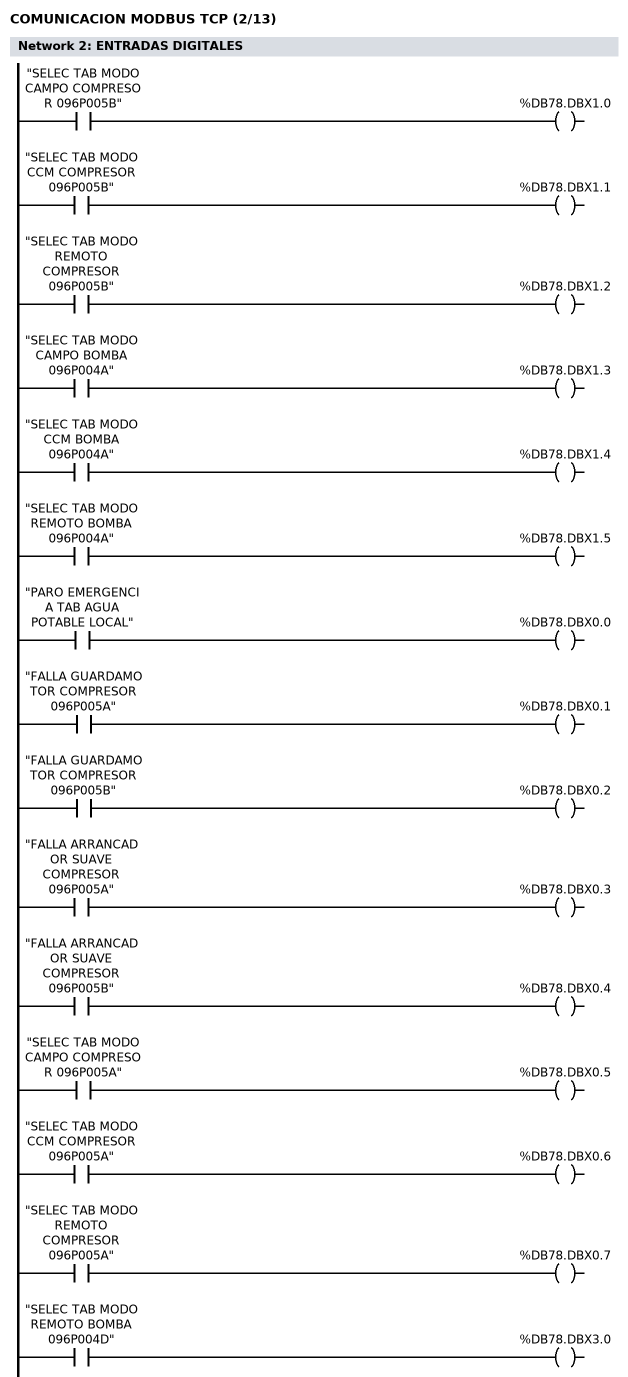
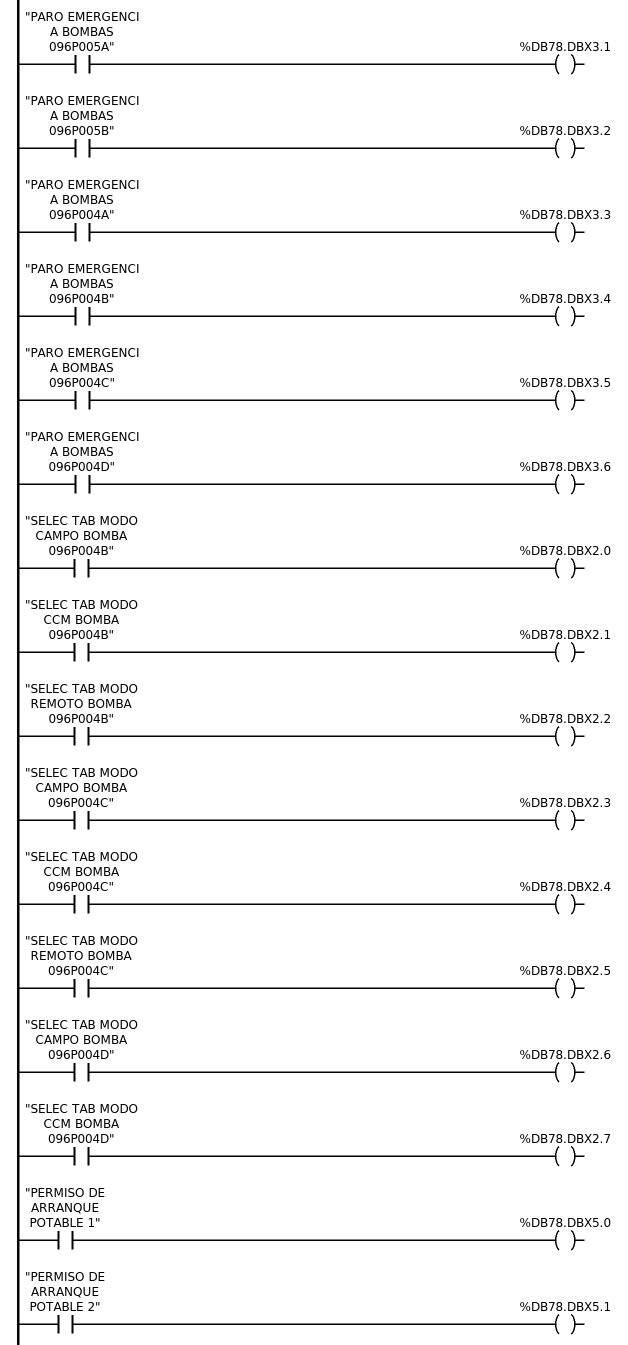
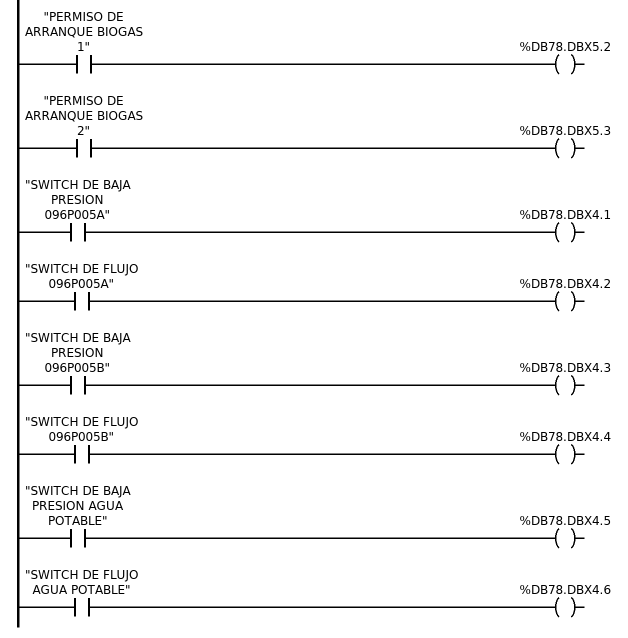
   RUNG wire#powerrail
      Contact( "SELEC TAB MODO CAMPO COMPRESOR 096P005B" )
      Coil( %DB78.DBX1.0 )
   END_RUNG
   RUNG wire#powerrail
      Contact( "SELEC TAB MODO CCM COMPRESOR 096P005B" )
      Coil( %DB78.DBX1.1 )
   END_RUNG
   RUNG wire#powerrail
      Contact( "SELEC TAB MODO REMOTO COMPRESOR 096P005B" )
      Coil( %DB78.DBX1.2 )
   END_RUNG
   RUNG wire#powerrail
      Contact( "SELEC TAB MODO CAMPO BOMBA 096P004A" )
      Coil( %DB78.DBX1.3 )
   END_RUNG
   RUNG wire#powerrail
      Contact( "SELEC TAB MODO CCM BOMBA 096P004A" )
      Coil( %DB78.DBX1.4 )
   END_RUNG
   RUNG wire#powerrail
      Contact( "SELEC TAB MODO REMOTO BOMBA 096P004A" )
      Coil( %DB78.DBX1.5 )
   END_RUNG
   RUNG wire#powerrail
      Contact( "PARO EMERGENCIA TAB AGUA POTABLE LOCAL" )
      Coil( %DB78.DBX0.0 )
   END_RUNG
   RUNG wire#powerrail
      Contact( "FALLA GUARDAMOTOR COMPRESOR 096P005A" )
      Coil( %DB78.DBX0.1 )
   END_RUNG
   RUNG wire#powerrail
      Contact( "FALLA GUARDAMOTOR COMPRESOR 096P005B" )
      Coil( %DB78.DBX0.2 )
   END_RUNG
   RUNG wire#powerrail
      Contact( "FALLA ARRANCADOR SUAVE COMPRESOR 096P005A" )
      Coil( %DB78.DBX0.3 )
   END_RUNG
   RUNG wire#powerrail
      Contact( "FALLA ARRANCADOR SUAVE COMPRESOR 096P005B" )
      Coil( %DB78.DBX0.4 )
   END_RUNG
   RUNG wire#powerrail
      Contact( "SELEC TAB MODO CAMPO COMPRESOR 096P005A" )
      Coil( %DB78.DBX0.5 )
   END_RUNG
   RUNG wire#powerrail
      Contact( "SELEC TAB MODO CCM COMPRESOR 096P005A" )
      Coil( %DB78.DBX0.6 )
   END_RUNG
   RUNG wire#powerrail
      Contact( "SELEC TAB MODO REMOTO COMPRESOR 096P005A" )
      Coil( %DB78.DBX0.7 )
   END_RUNG
   RUNG wire#powerrail
      Contact( "SELEC TAB MODO REMOTO BOMBA 096P004D" )
      Coil( %DB78.DBX3.0 )
   END_RUNG
   RUNG wire#powerrail
      Contact( "PARO EMERGENCIA BOMBAS 096P005A" )
      Coil( %DB78.DBX3.1 )
   END_RUNG
   RUNG wire#powerrail
      Contact( "PARO EMERGENCIA BOMBAS 096P005B" )
      Coil( %DB78.DBX3.2 )
   END_RUNG
   RUNG wire#powerrail
      Contact( "PARO EMERGENCIA BOMBAS 096P004A" )
      Coil( %DB78.DBX3.3 )
   END_RUNG
   RUNG wire#powerrail
      Contact( "PARO EMERGENCIA BOMBAS 096P004B" )
      Coil( %DB78.DBX3.4 )
   END_RUNG
   RUNG wire#powerrail
      Contact( "PARO EMERGENCIA BOMBAS 096P004C" )
      Coil( %DB78.DBX3.5 )
   END_RUNG
   RUNG wire#powerrail
      Contact( "PARO EMERGENCIA BOMBAS 096P004D" )
      Coil( %DB78.DBX3.6 )
   END_RUNG
   RUNG wire#powerrail
      Contact( "SELEC TAB MODO CAMPO BOMBA 096P004B" )
      Coil( %DB78.DBX2.0 )
   END_RUNG
   RUNG wire#powerrail
      Contact( "SELEC TAB MODO CCM BOMBA 096P004B" )
      Coil( %DB78.DBX2.1 )
   END_RUNG
   RUNG wire#powerrail
      Contact( "SELEC TAB MODO REMOTO BOMBA 096P004B" )
      Coil( %DB78.DBX2.2 )
   END_RUNG
   RUNG wire#powerrail
      Contact( "SELEC TAB MODO CAMPO BOMBA 096P004C" )
      Coil( %DB78.DBX2.3 )
   END_RUNG
   RUNG wire#powerrail
      Contact( "SELEC TAB MODO CCM BOMBA 096P004C" )
      Coil( %DB78.DBX2.4 )
   END_RUNG
   RUNG wire#powerrail
      Contact( "SELEC TAB MODO REMOTO BOMBA 096P004C" )
      Coil( %DB78.DBX2.5 )
   END_RUNG
   RUNG wire#powerrail
      Contact( "SELEC TAB MODO CAMPO BOMBA 096P004D" )
      Coil( %DB78.DBX2.6 )
   END_RUNG
   RUNG wire#powerrail
      Contact( "SELEC TAB MODO CCM BOMBA 096P004D" )
      Coil( %DB78.DBX2.7 )
   END_RUNG
   RUNG wire#powerrail
      Contact( "PERMISO DE ARRANQUE POTABLE 1" )
      Coil( %DB78.DBX5.0 )
   END_RUNG
   RUNG wire#powerrail
      Contact( "PERMISO DE ARRANQUE POTABLE 2" )
      Coil( %DB78.DBX5.1 )
   END_RUNG
   RUNG wire#powerrail
      Contact( "PERMISO DE ARRANQUE BIOGAS 1" )
      Coil( %DB78.DBX5.2 )
   END_RUNG
   RUNG wire#powerrail
      Contact( "PERMISO DE ARRANQUE BIOGAS 2" )
      Coil( %DB78.DBX5.3 )
   END_RUNG
   RUNG wire#powerrail
      Contact( "SWITCH DE BAJA PRESION 096P005A" )
      Coil( %DB78.DBX4.1 )
   END_RUNG
   RUNG wire#powerrail
      Contact( "SWITCH DE FLUJO 096P005A" )
      Coil( %DB78.DBX4.2 )
   END_RUNG
   RUNG wire#powerrail
      Contact( "SWITCH DE BAJA PRESION 096P005B" )
      Coil( %DB78.DBX4.3 )
   END_RUNG
   RUNG wire#powerrail
      Contact( "SWITCH DE FLUJO 096P005B" )
      Coil( %DB78.DBX4.4 )
   END_RUNG
   RUNG wire#powerrail
      Contact( "SWITCH DE BAJA PRESION AGUA POTABLE" )
      Coil( %DB78.DBX4.5 )
   END_RUNG
   RUNG wire#powerrail
      Contact( "SWITCH DE FLUJO AGUA POTABLE" )
      Coil( %DB78.DBX4.6 )
   END_RUNG
   // the same network as SCL:
   %DB78.DBX1.0 := "SELEC TAB MODO CAMPO COMPRESOR 096P005B";
   %DB78.DBX1.1 := "SELEC TAB MODO CCM COMPRESOR 096P005B";
   %DB78.DBX1.2 := "SELEC TAB MODO REMOTO COMPRESOR 096P005B";
   %DB78.DBX1.3 := "SELEC TAB MODO CAMPO BOMBA 096P004A";
   %DB78.DBX1.4 := "SELEC TAB MODO CCM BOMBA 096P004A";
   %DB78.DBX1.5 := "SELEC TAB MODO REMOTO BOMBA 096P004A";
   %DB78.DBX0.0 := "PARO EMERGENCIA TAB AGUA POTABLE LOCAL";
   %DB78.DBX0.1 := "FALLA GUARDAMOTOR COMPRESOR 096P005A";
   %DB78.DBX0.2 := "FALLA GUARDAMOTOR COMPRESOR 096P005B";
   %DB78.DBX0.3 := "FALLA ARRANCADOR SUAVE COMPRESOR 096P005A";
   %DB78.DBX0.4 := "FALLA ARRANCADOR SUAVE COMPRESOR 096P005B";
   %DB78.DBX0.5 := "SELEC TAB MODO CAMPO COMPRESOR 096P005A";
   %DB78.DBX0.6 := "SELEC TAB MODO CCM COMPRESOR 096P005A";
   %DB78.DBX0.7 := "SELEC TAB MODO REMOTO COMPRESOR 096P005A";
   %DB78.DBX3.0 := "SELEC TAB MODO REMOTO BOMBA 096P004D";
   %DB78.DBX3.1 := "PARO EMERGENCIA BOMBAS 096P005A";
   %DB78.DBX3.2 := "PARO EMERGENCIA BOMBAS 096P005B";
   %DB78.DBX3.3 := "PARO EMERGENCIA BOMBAS 096P004A";
   %DB78.DBX3.4 := "PARO EMERGENCIA BOMBAS 096P004B";
   %DB78.DBX3.5 := "PARO EMERGENCIA BOMBAS 096P004C";
   %DB78.DBX3.6 := "PARO EMERGENCIA BOMBAS 096P004D";
   %DB78.DBX2.0 := "SELEC TAB MODO CAMPO BOMBA 096P004B";
   %DB78.DBX2.1 := "SELEC TAB MODO CCM BOMBA 096P004B";
   %DB78.DBX2.2 := "SELEC TAB MODO REMOTO BOMBA 096P004B";
   %DB78.DBX2.3 := "SELEC TAB MODO CAMPO BOMBA 096P004C";
   %DB78.DBX2.4 := "SELEC TAB MODO CCM BOMBA 096P004C";
   %DB78.DBX2.5 := "SELEC TAB MODO REMOTO BOMBA 096P004C";
   %DB78.DBX2.6 := "SELEC TAB MODO CAMPO BOMBA 096P004D";
   %DB78.DBX2.7 := "SELEC TAB MODO CCM BOMBA 096P004D";
   %DB78.DBX5.0 := "PERMISO DE ARRANQUE POTABLE 1";
   %DB78.DBX5.1 := "PERMISO DE ARRANQUE POTABLE 2";
   %DB78.DBX5.2 := "PERMISO DE ARRANQUE BIOGAS 1";
   %DB78.DBX5.3 := "PERMISO DE ARRANQUE BIOGAS 2";
   %DB78.DBX4.1 := "SWITCH DE BAJA PRESION 096P005A";
   %DB78.DBX4.2 := "SWITCH DE FLUJO 096P005A";
   %DB78.DBX4.3 := "SWITCH DE BAJA PRESION 096P005B";
   %DB78.DBX4.4 := "SWITCH DE FLUJO 096P005B";
   %DB78.DBX4.5 := "SWITCH DE BAJA PRESION AGUA POTABLE";
   %DB78.DBX4.6 := "SWITCH DE FLUJO AGUA POTABLE";
END_REGION

REGION Network 3: SALIDAS DIGITALES
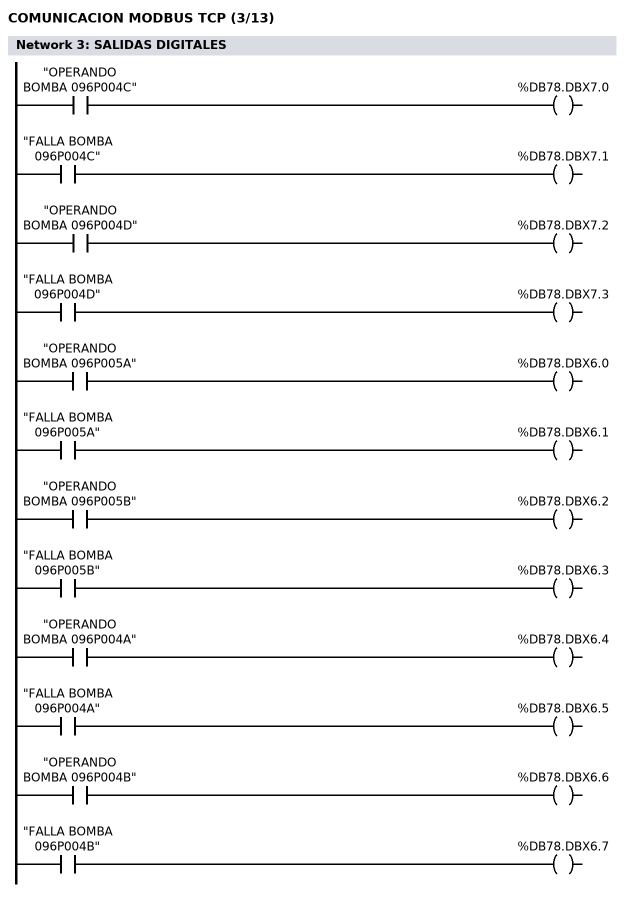
   RUNG wire#powerrail
      Contact( "OPERANDO BOMBA 096P004C" )
      Coil( %DB78.DBX7.0 )
   END_RUNG
   RUNG wire#powerrail
      Contact( "FALLA BOMBA 096P004C" )
      Coil( %DB78.DBX7.1 )
   END_RUNG
   RUNG wire#powerrail
      Contact( "OPERANDO BOMBA 096P004D" )
      Coil( %DB78.DBX7.2 )
   END_RUNG
   RUNG wire#powerrail
      Contact( "FALLA BOMBA 096P004D" )
      Coil( %DB78.DBX7.3 )
   END_RUNG
   RUNG wire#powerrail
      Contact( "OPERANDO BOMBA 096P005A" )
      Coil( %DB78.DBX6.0 )
   END_RUNG
   RUNG wire#powerrail
      Contact( "FALLA BOMBA 096P005A" )
      Coil( %DB78.DBX6.1 )
   END_RUNG
   RUNG wire#powerrail
      Contact( "OPERANDO BOMBA 096P005B" )
      Coil( %DB78.DBX6.2 )
   END_RUNG
   RUNG wire#powerrail
      Contact( "FALLA BOMBA 096P005B" )
      Coil( %DB78.DBX6.3 )
   END_RUNG
   RUNG wire#powerrail
      Contact( "OPERANDO BOMBA 096P004A" )
      Coil( %DB78.DBX6.4 )
   END_RUNG
   RUNG wire#powerrail
      Contact( "FALLA BOMBA 096P004A" )
      Coil( %DB78.DBX6.5 )
   END_RUNG
   RUNG wire#powerrail
      Contact( "OPERANDO BOMBA 096P004B" )
      Coil( %DB78.DBX6.6 )
   END_RUNG
   RUNG wire#powerrail
      Contact( "FALLA BOMBA 096P004B" )
      Coil( %DB78.DBX6.7 )
   END_RUNG
   // the same network as SCL:
   %DB78.DBX7.0 := "OPERANDO BOMBA 096P004C";
   %DB78.DBX7.1 := "FALLA BOMBA 096P004C";
   %DB78.DBX7.2 := "OPERANDO BOMBA 096P004D";
   %DB78.DBX7.3 := "FALLA BOMBA 096P004D";
   %DB78.DBX6.0 := "OPERANDO BOMBA 096P005A";
   %DB78.DBX6.1 := "FALLA BOMBA 096P005A";
   %DB78.DBX6.2 := "OPERANDO BOMBA 096P005B";
   %DB78.DBX6.3 := "FALLA BOMBA 096P005B";
   %DB78.DBX6.4 := "OPERANDO BOMBA 096P004A";
   %DB78.DBX6.5 := "FALLA BOMBA 096P004A";
   %DB78.DBX6.6 := "OPERANDO BOMBA 096P004B";
   %DB78.DBX6.7 := "FALLA BOMBA 096P004B";
END_REGION

REGION Network 4: SET POINT
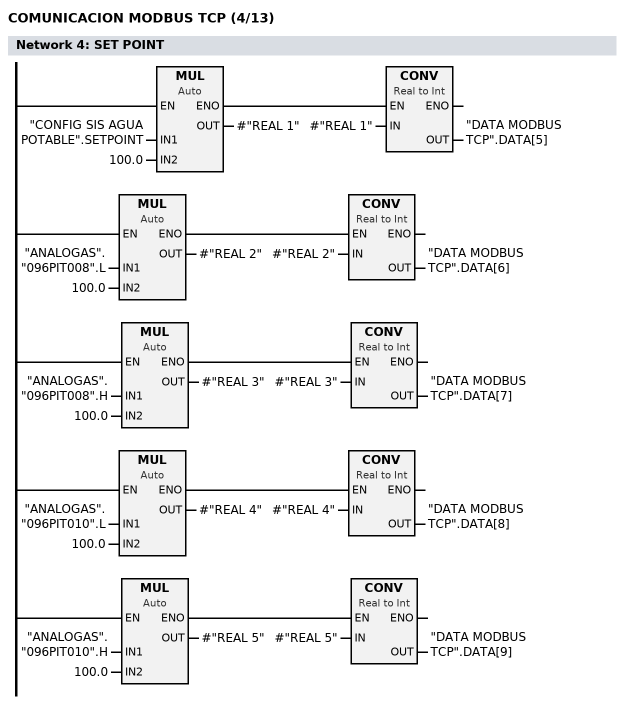
   RUNG wire#powerrail
      Mul(in1 := "CONFIG SIS AGUA POTABLE".SETPOINT, in2 := 100.0, out => #"REAL 1")
      { S7_Templates := "[SrcType := Real, DestType := Int]" } Convert(in := #"REAL 1", out => "DATA MODBUS TCP".DATA[5])
   END_RUNG
   RUNG wire#powerrail
      Mul(in1 := "ANALOGAS"."096PIT008".L, in2 := 100.0, out => #"REAL 2")
      { S7_Templates := "[SrcType := Real, DestType := Int]" } Convert(in := #"REAL 2", out => "DATA MODBUS TCP".DATA[6])
   END_RUNG
   RUNG wire#powerrail
      Mul(in1 := "ANALOGAS"."096PIT008".H, in2 := 100.0, out => #"REAL 3")
      { S7_Templates := "[SrcType := Real, DestType := Int]" } Convert(in := #"REAL 3", out => "DATA MODBUS TCP".DATA[7])
   END_RUNG
   RUNG wire#powerrail
      Mul(in1 := "ANALOGAS"."096PIT010".L, in2 := 100.0, out => #"REAL 4")
      { S7_Templates := "[SrcType := Real, DestType := Int]" } Convert(in := #"REAL 4", out => "DATA MODBUS TCP".DATA[8])
   END_RUNG
   RUNG wire#powerrail
      Mul(in1 := "ANALOGAS"."096PIT010".H, in2 := 100.0, out => #"REAL 5")
      { S7_Templates := "[SrcType := Real, DestType := Int]" } Convert(in := #"REAL 5", out => "DATA MODBUS TCP".DATA[9])
   END_RUNG
   // the same network as SCL:
   #"REAL 1" := "CONFIG SIS AGUA POTABLE".SETPOINT * 100.0;
   "DATA MODBUS TCP".DATA[5] := REAL_TO_INT(#"REAL 1");
   #"REAL 2" := "ANALOGAS"."096PIT008".L * 100.0;
   "DATA MODBUS TCP".DATA[6] := REAL_TO_INT(#"REAL 2");
   #"REAL 3" := "ANALOGAS"."096PIT008".H * 100.0;
   "DATA MODBUS TCP".DATA[7] := REAL_TO_INT(#"REAL 3");
   #"REAL 4" := "ANALOGAS"."096PIT010".L * 100.0;
   "DATA MODBUS TCP".DATA[8] := REAL_TO_INT(#"REAL 4");
   #"REAL 5" := "ANALOGAS"."096PIT010".H * 100.0;
   "DATA MODBUS TCP".DATA[9] := REAL_TO_INT(#"REAL 5");
END_REGION

REGION Network 5: ANALOGAS
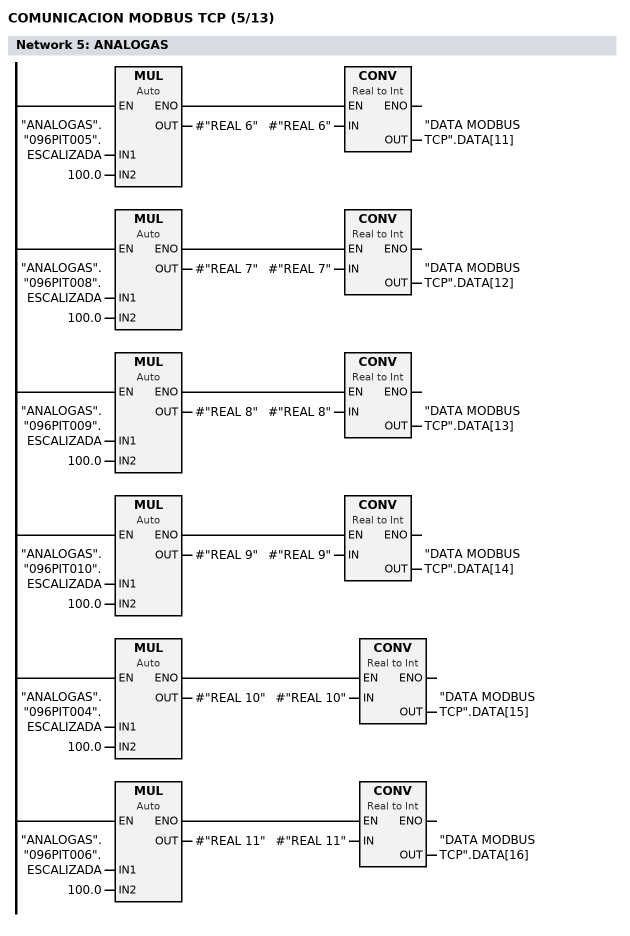
   RUNG wire#powerrail
      Mul(in1 := "ANALOGAS"."096PIT005".ESCALIZADA, in2 := 100.0, out => #"REAL 6")
      { S7_Templates := "[SrcType := Real, DestType := Int]" } Convert(in := #"REAL 6", out => "DATA MODBUS TCP".DATA[11])
   END_RUNG
   RUNG wire#powerrail
      Mul(in1 := "ANALOGAS"."096PIT008".ESCALIZADA, in2 := 100.0, out => #"REAL 7")
      { S7_Templates := "[SrcType := Real, DestType := Int]" } Convert(in := #"REAL 7", out => "DATA MODBUS TCP".DATA[12])
   END_RUNG
   RUNG wire#powerrail
      Mul(in1 := "ANALOGAS"."096PIT009".ESCALIZADA, in2 := 100.0, out => #"REAL 8")
      { S7_Templates := "[SrcType := Real, DestType := Int]" } Convert(in := #"REAL 8", out => "DATA MODBUS TCP".DATA[13])
   END_RUNG
   RUNG wire#powerrail
      Mul(in1 := "ANALOGAS"."096PIT010".ESCALIZADA, in2 := 100.0, out => #"REAL 9")
      { S7_Templates := "[SrcType := Real, DestType := Int]" } Convert(in := #"REAL 9", out => "DATA MODBUS TCP".DATA[14])
   END_RUNG
   RUNG wire#powerrail
      Mul(in1 := "ANALOGAS"."096PIT004".ESCALIZADA, in2 := 100.0, out => #"REAL 10")
      { S7_Templates := "[SrcType := Real, DestType := Int]" } Convert(in := #"REAL 10", out => "DATA MODBUS TCP".DATA[15])
   END_RUNG
   RUNG wire#powerrail
      Mul(in1 := "ANALOGAS"."096PIT006".ESCALIZADA, in2 := 100.0, out => #"REAL 11")
      { S7_Templates := "[SrcType := Real, DestType := Int]" } Convert(in := #"REAL 11", out => "DATA MODBUS TCP".DATA[16])
   END_RUNG
   // the same network as SCL:
   #"REAL 6" := "ANALOGAS"."096PIT005".ESCALIZADA * 100.0;
   "DATA MODBUS TCP".DATA[11] := REAL_TO_INT(#"REAL 6");
   #"REAL 7" := "ANALOGAS"."096PIT008".ESCALIZADA * 100.0;
   "DATA MODBUS TCP".DATA[12] := REAL_TO_INT(#"REAL 7");
   #"REAL 8" := "ANALOGAS"."096PIT009".ESCALIZADA * 100.0;
   "DATA MODBUS TCP".DATA[13] := REAL_TO_INT(#"REAL 8");
   #"REAL 9" := "ANALOGAS"."096PIT010".ESCALIZADA * 100.0;
   "DATA MODBUS TCP".DATA[14] := REAL_TO_INT(#"REAL 9");
   #"REAL 10" := "ANALOGAS"."096PIT004".ESCALIZADA * 100.0;
   "DATA MODBUS TCP".DATA[15] := REAL_TO_INT(#"REAL 10");
   #"REAL 11" := "ANALOGAS"."096PIT006".ESCALIZADA * 100.0;
   "DATA MODBUS TCP".DATA[16] := REAL_TO_INT(#"REAL 11");
END_REGION

REGION Network 6: ORDEN DE CAMBIO DE MODO BOMBA 5A
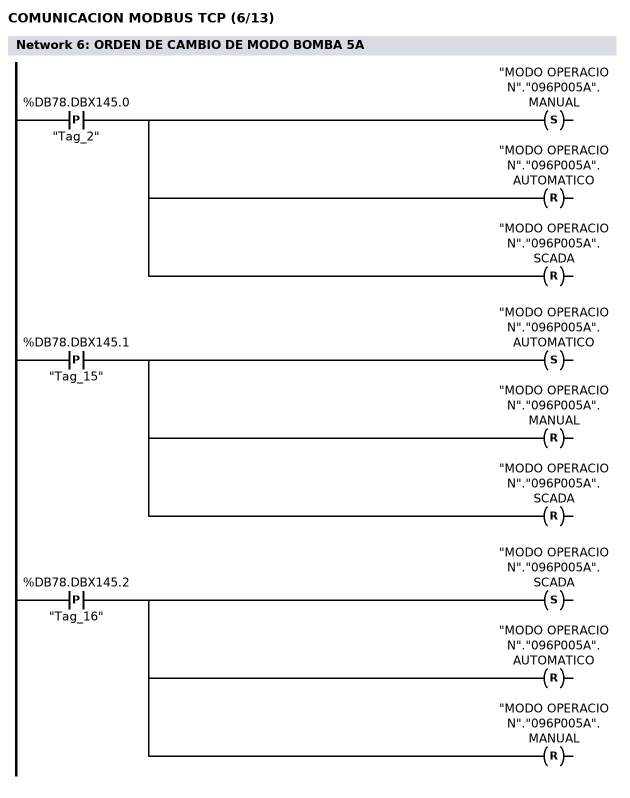
   RUNG wire#powerrail
      P_Contact(operand := %DB78.DBX145.0, bit := "Tag_2")
      wire#w1
      S_Coil( "MODO OPERACION"."096P005A".MANUAL )
   END_RUNG
   RUNG wire#w1
      R_Coil( "MODO OPERACION"."096P005A".AUTOMATICO )
   END_RUNG
   RUNG wire#w1
      R_Coil( "MODO OPERACION"."096P005A".SCADA )
   END_RUNG
   RUNG wire#powerrail
      P_Contact(operand := %DB78.DBX145.1, bit := "Tag_15")
      wire#w2
      S_Coil( "MODO OPERACION"."096P005A".AUTOMATICO )
   END_RUNG
   RUNG wire#w2
      R_Coil( "MODO OPERACION"."096P005A".MANUAL )
   END_RUNG
   RUNG wire#w2
      R_Coil( "MODO OPERACION"."096P005A".SCADA )
   END_RUNG
   RUNG wire#powerrail
      P_Contact(operand := %DB78.DBX145.2, bit := "Tag_16")
      wire#w3
      S_Coil( "MODO OPERACION"."096P005A".SCADA )
   END_RUNG
   RUNG wire#w3
      R_Coil( "MODO OPERACION"."096P005A".AUTOMATICO )
   END_RUNG
   RUNG wire#w3
      R_Coil( "MODO OPERACION"."096P005A".MANUAL )
   END_RUNG
   // the same network as SCL:
   #_w1 := %DB78.DBX145.0 AND NOT "Tag_2";   // rising edge of %DB78.DBX145.0
   "Tag_2" := %DB78.DBX145.0;
   IF #_w1 THEN
       "MODO OPERACION"."096P005A".MANUAL := TRUE;
       "MODO OPERACION"."096P005A".AUTOMATICO := FALSE;
       "MODO OPERACION"."096P005A".SCADA := FALSE;
   END_IF;
   #_w2 := %DB78.DBX145.1 AND NOT "Tag_15";   // rising edge of %DB78.DBX145.1
   "Tag_15" := %DB78.DBX145.1;
   IF #_w2 THEN
       "MODO OPERACION"."096P005A".AUTOMATICO := TRUE;
       "MODO OPERACION"."096P005A".MANUAL := FALSE;
       "MODO OPERACION"."096P005A".SCADA := FALSE;
   END_IF;
   #_w3 := %DB78.DBX145.2 AND NOT "Tag_16";   // rising edge of %DB78.DBX145.2
   "Tag_16" := %DB78.DBX145.2;
   IF #_w3 THEN
       "MODO OPERACION"."096P005A".SCADA := TRUE;
       "MODO OPERACION"."096P005A".AUTOMATICO := FALSE;
       "MODO OPERACION"."096P005A".MANUAL := FALSE;
   END_IF;
END_REGION

REGION Network 7: ORDEN DE CAMBIO DE MODO BOMBA 5B
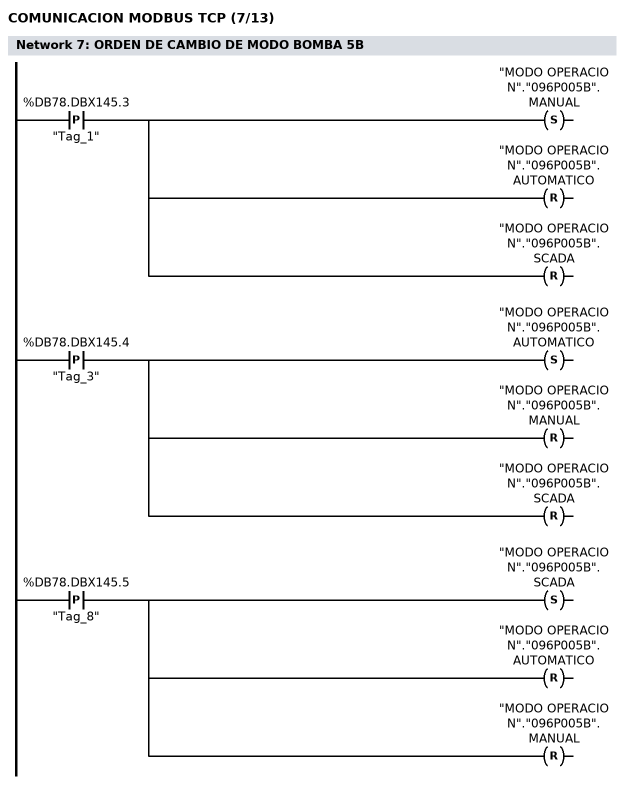
   RUNG wire#powerrail
      P_Contact(operand := %DB78.DBX145.3, bit := "Tag_1")
      wire#w1
      S_Coil( "MODO OPERACION"."096P005B".MANUAL )
   END_RUNG
   RUNG wire#w1
      R_Coil( "MODO OPERACION"."096P005B".AUTOMATICO )
   END_RUNG
   RUNG wire#w1
      R_Coil( "MODO OPERACION"."096P005B".SCADA )
   END_RUNG
   RUNG wire#powerrail
      P_Contact(operand := %DB78.DBX145.4, bit := "Tag_3")
      wire#w2
      S_Coil( "MODO OPERACION"."096P005B".AUTOMATICO )
   END_RUNG
   RUNG wire#w2
      R_Coil( "MODO OPERACION"."096P005B".MANUAL )
   END_RUNG
   RUNG wire#w2
      R_Coil( "MODO OPERACION"."096P005B".SCADA )
   END_RUNG
   RUNG wire#powerrail
      P_Contact(operand := %DB78.DBX145.5, bit := "Tag_8")
      wire#w3
      S_Coil( "MODO OPERACION"."096P005B".SCADA )
   END_RUNG
   RUNG wire#w3
      R_Coil( "MODO OPERACION"."096P005B".AUTOMATICO )
   END_RUNG
   RUNG wire#w3
      R_Coil( "MODO OPERACION"."096P005B".MANUAL )
   END_RUNG
   // the same network as SCL:
   #_w1 := %DB78.DBX145.3 AND NOT "Tag_1";   // rising edge of %DB78.DBX145.3
   "Tag_1" := %DB78.DBX145.3;
   IF #_w1 THEN
       "MODO OPERACION"."096P005B".MANUAL := TRUE;
       "MODO OPERACION"."096P005B".AUTOMATICO := FALSE;
       "MODO OPERACION"."096P005B".SCADA := FALSE;
   END_IF;
   #_w2 := %DB78.DBX145.4 AND NOT "Tag_3";   // rising edge of %DB78.DBX145.4
   "Tag_3" := %DB78.DBX145.4;
   IF #_w2 THEN
       "MODO OPERACION"."096P005B".AUTOMATICO := TRUE;
       "MODO OPERACION"."096P005B".MANUAL := FALSE;
       "MODO OPERACION"."096P005B".SCADA := FALSE;
   END_IF;
   #_w3 := %DB78.DBX145.5 AND NOT "Tag_8";   // rising edge of %DB78.DBX145.5
   "Tag_8" := %DB78.DBX145.5;
   IF #_w3 THEN
       "MODO OPERACION"."096P005B".SCADA := TRUE;
       "MODO OPERACION"."096P005B".AUTOMATICO := FALSE;
       "MODO OPERACION"."096P005B".MANUAL := FALSE;
   END_IF;
END_REGION

REGION Network 8: ORDEN DE CAMBIO DE MODO BOMBA 4A
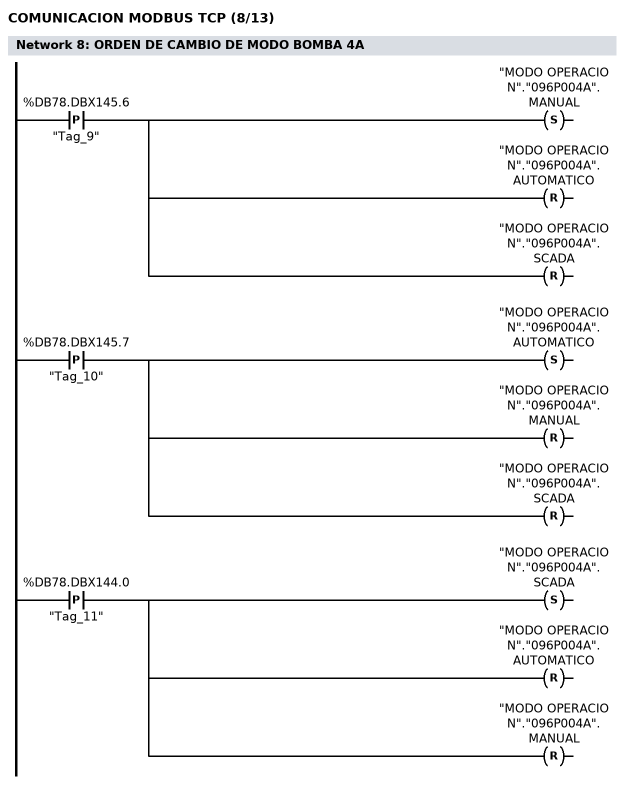
   RUNG wire#powerrail
      P_Contact(operand := %DB78.DBX145.6, bit := "Tag_9")
      wire#w1
      S_Coil( "MODO OPERACION"."096P004A".MANUAL )
   END_RUNG
   RUNG wire#w1
      R_Coil( "MODO OPERACION"."096P004A".AUTOMATICO )
   END_RUNG
   RUNG wire#w1
      R_Coil( "MODO OPERACION"."096P004A".SCADA )
   END_RUNG
   RUNG wire#powerrail
      P_Contact(operand := %DB78.DBX145.7, bit := "Tag_10")
      wire#w2
      S_Coil( "MODO OPERACION"."096P004A".AUTOMATICO )
   END_RUNG
   RUNG wire#w2
      R_Coil( "MODO OPERACION"."096P004A".MANUAL )
   END_RUNG
   RUNG wire#w2
      R_Coil( "MODO OPERACION"."096P004A".SCADA )
   END_RUNG
   RUNG wire#powerrail
      P_Contact(operand := %DB78.DBX144.0, bit := "Tag_11")
      wire#w3
      S_Coil( "MODO OPERACION"."096P004A".SCADA )
   END_RUNG
   RUNG wire#w3
      R_Coil( "MODO OPERACION"."096P004A".AUTOMATICO )
   END_RUNG
   RUNG wire#w3
      R_Coil( "MODO OPERACION"."096P004A".MANUAL )
   END_RUNG
   // the same network as SCL:
   #_w1 := %DB78.DBX145.6 AND NOT "Tag_9";   // rising edge of %DB78.DBX145.6
   "Tag_9" := %DB78.DBX145.6;
   IF #_w1 THEN
       "MODO OPERACION"."096P004A".MANUAL := TRUE;
       "MODO OPERACION"."096P004A".AUTOMATICO := FALSE;
       "MODO OPERACION"."096P004A".SCADA := FALSE;
   END_IF;
   #_w2 := %DB78.DBX145.7 AND NOT "Tag_10";   // rising edge of %DB78.DBX145.7
   "Tag_10" := %DB78.DBX145.7;
   IF #_w2 THEN
       "MODO OPERACION"."096P004A".AUTOMATICO := TRUE;
       "MODO OPERACION"."096P004A".MANUAL := FALSE;
       "MODO OPERACION"."096P004A".SCADA := FALSE;
   END_IF;
   #_w3 := %DB78.DBX144.0 AND NOT "Tag_11";   // rising edge of %DB78.DBX144.0
   "Tag_11" := %DB78.DBX144.0;
   IF #_w3 THEN
       "MODO OPERACION"."096P004A".SCADA := TRUE;
       "MODO OPERACION"."096P004A".AUTOMATICO := FALSE;
       "MODO OPERACION"."096P004A".MANUAL := FALSE;
   END_IF;
END_REGION

REGION Network 9: ORDEN DE CAMBIO DE MODO BOMBA 4B
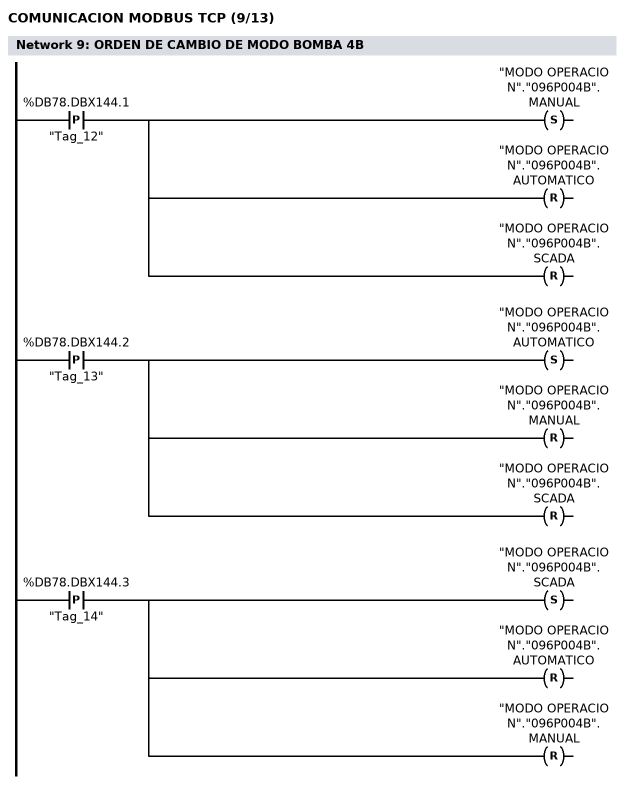
   RUNG wire#powerrail
      P_Contact(operand := %DB78.DBX144.1, bit := "Tag_12")
      wire#w1
      S_Coil( "MODO OPERACION"."096P004B".MANUAL )
   END_RUNG
   RUNG wire#w1
      R_Coil( "MODO OPERACION"."096P004B".AUTOMATICO )
   END_RUNG
   RUNG wire#w1
      R_Coil( "MODO OPERACION"."096P004B".SCADA )
   END_RUNG
   RUNG wire#powerrail
      P_Contact(operand := %DB78.DBX144.2, bit := "Tag_13")
      wire#w2
      S_Coil( "MODO OPERACION"."096P004B".AUTOMATICO )
   END_RUNG
   RUNG wire#w2
      R_Coil( "MODO OPERACION"."096P004B".MANUAL )
   END_RUNG
   RUNG wire#w2
      R_Coil( "MODO OPERACION"."096P004B".SCADA )
   END_RUNG
   RUNG wire#powerrail
      P_Contact(operand := %DB78.DBX144.3, bit := "Tag_14")
      wire#w3
      S_Coil( "MODO OPERACION"."096P004B".SCADA )
   END_RUNG
   RUNG wire#w3
      R_Coil( "MODO OPERACION"."096P004B".AUTOMATICO )
   END_RUNG
   RUNG wire#w3
      R_Coil( "MODO OPERACION"."096P004B".MANUAL )
   END_RUNG
   // the same network as SCL:
   #_w1 := %DB78.DBX144.1 AND NOT "Tag_12";   // rising edge of %DB78.DBX144.1
   "Tag_12" := %DB78.DBX144.1;
   IF #_w1 THEN
       "MODO OPERACION"."096P004B".MANUAL := TRUE;
       "MODO OPERACION"."096P004B".AUTOMATICO := FALSE;
       "MODO OPERACION"."096P004B".SCADA := FALSE;
   END_IF;
   #_w2 := %DB78.DBX144.2 AND NOT "Tag_13";   // rising edge of %DB78.DBX144.2
   "Tag_13" := %DB78.DBX144.2;
   IF #_w2 THEN
       "MODO OPERACION"."096P004B".AUTOMATICO := TRUE;
       "MODO OPERACION"."096P004B".MANUAL := FALSE;
       "MODO OPERACION"."096P004B".SCADA := FALSE;
   END_IF;
   #_w3 := %DB78.DBX144.3 AND NOT "Tag_14";   // rising edge of %DB78.DBX144.3
   "Tag_14" := %DB78.DBX144.3;
   IF #_w3 THEN
       "MODO OPERACION"."096P004B".SCADA := TRUE;
       "MODO OPERACION"."096P004B".AUTOMATICO := FALSE;
       "MODO OPERACION"."096P004B".MANUAL := FALSE;
   END_IF;
END_REGION

REGION Network 10: ORDEN DE CAMBIO DE MODO BOMBA 4C
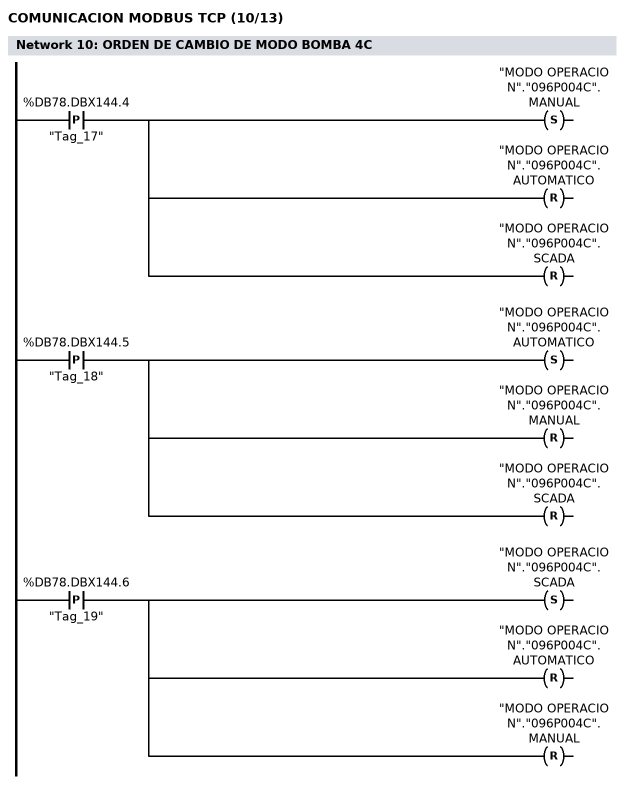
   RUNG wire#powerrail
      P_Contact(operand := %DB78.DBX144.4, bit := "Tag_17")
      wire#w1
      S_Coil( "MODO OPERACION"."096P004C".MANUAL )
   END_RUNG
   RUNG wire#w1
      R_Coil( "MODO OPERACION"."096P004C".AUTOMATICO )
   END_RUNG
   RUNG wire#w1
      R_Coil( "MODO OPERACION"."096P004C".SCADA )
   END_RUNG
   RUNG wire#powerrail
      P_Contact(operand := %DB78.DBX144.5, bit := "Tag_18")
      wire#w2
      S_Coil( "MODO OPERACION"."096P004C".AUTOMATICO )
   END_RUNG
   RUNG wire#w2
      R_Coil( "MODO OPERACION"."096P004C".MANUAL )
   END_RUNG
   RUNG wire#w2
      R_Coil( "MODO OPERACION"."096P004C".SCADA )
   END_RUNG
   RUNG wire#powerrail
      P_Contact(operand := %DB78.DBX144.6, bit := "Tag_19")
      wire#w3
      S_Coil( "MODO OPERACION"."096P004C".SCADA )
   END_RUNG
   RUNG wire#w3
      R_Coil( "MODO OPERACION"."096P004C".AUTOMATICO )
   END_RUNG
   RUNG wire#w3
      R_Coil( "MODO OPERACION"."096P004C".MANUAL )
   END_RUNG
   // the same network as SCL:
   #_w1 := %DB78.DBX144.4 AND NOT "Tag_17";   // rising edge of %DB78.DBX144.4
   "Tag_17" := %DB78.DBX144.4;
   IF #_w1 THEN
       "MODO OPERACION"."096P004C".MANUAL := TRUE;
       "MODO OPERACION"."096P004C".AUTOMATICO := FALSE;
       "MODO OPERACION"."096P004C".SCADA := FALSE;
   END_IF;
   #_w2 := %DB78.DBX144.5 AND NOT "Tag_18";   // rising edge of %DB78.DBX144.5
   "Tag_18" := %DB78.DBX144.5;
   IF #_w2 THEN
       "MODO OPERACION"."096P004C".AUTOMATICO := TRUE;
       "MODO OPERACION"."096P004C".MANUAL := FALSE;
       "MODO OPERACION"."096P004C".SCADA := FALSE;
   END_IF;
   #_w3 := %DB78.DBX144.6 AND NOT "Tag_19";   // rising edge of %DB78.DBX144.6
   "Tag_19" := %DB78.DBX144.6;
   IF #_w3 THEN
       "MODO OPERACION"."096P004C".SCADA := TRUE;
       "MODO OPERACION"."096P004C".AUTOMATICO := FALSE;
       "MODO OPERACION"."096P004C".MANUAL := FALSE;
   END_IF;
END_REGION

REGION Network 11: ORDEN DE CAMBIO DE MODO BOMBA 4D
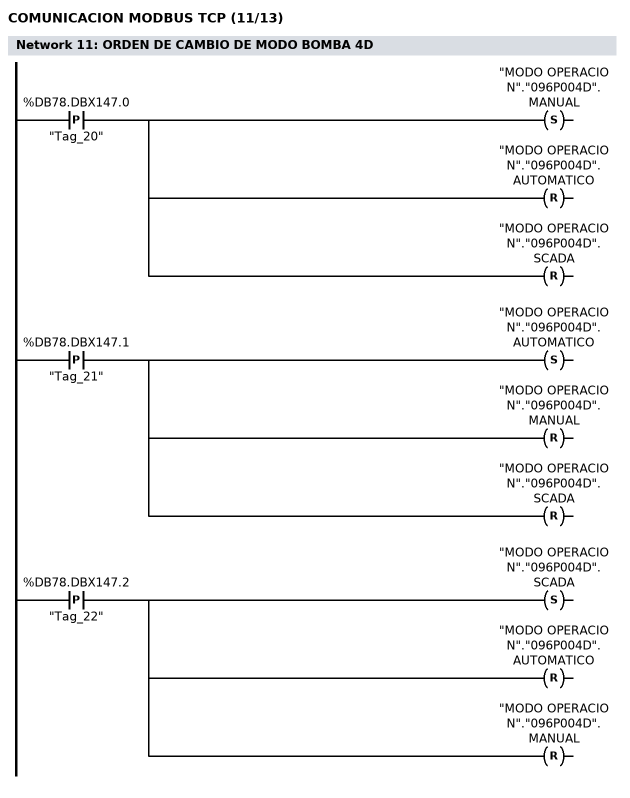
   RUNG wire#powerrail
      P_Contact(operand := %DB78.DBX147.0, bit := "Tag_20")
      wire#w1
      S_Coil( "MODO OPERACION"."096P004D".MANUAL )
   END_RUNG
   RUNG wire#w1
      R_Coil( "MODO OPERACION"."096P004D".AUTOMATICO )
   END_RUNG
   RUNG wire#w1
      R_Coil( "MODO OPERACION"."096P004D".SCADA )
   END_RUNG
   RUNG wire#powerrail
      P_Contact(operand := %DB78.DBX147.1, bit := "Tag_21")
      wire#w2
      S_Coil( "MODO OPERACION"."096P004D".AUTOMATICO )
   END_RUNG
   RUNG wire#w2
      R_Coil( "MODO OPERACION"."096P004D".MANUAL )
   END_RUNG
   RUNG wire#w2
      R_Coil( "MODO OPERACION"."096P004D".SCADA )
   END_RUNG
   RUNG wire#powerrail
      P_Contact(operand := %DB78.DBX147.2, bit := "Tag_22")
      wire#w3
      S_Coil( "MODO OPERACION"."096P004D".SCADA )
   END_RUNG
   RUNG wire#w3
      R_Coil( "MODO OPERACION"."096P004D".AUTOMATICO )
   END_RUNG
   RUNG wire#w3
      R_Coil( "MODO OPERACION"."096P004D".MANUAL )
   END_RUNG
   // the same network as SCL:
   #_w1 := %DB78.DBX147.0 AND NOT "Tag_20";   // rising edge of %DB78.DBX147.0
   "Tag_20" := %DB78.DBX147.0;
   IF #_w1 THEN
       "MODO OPERACION"."096P004D".MANUAL := TRUE;
       "MODO OPERACION"."096P004D".AUTOMATICO := FALSE;
       "MODO OPERACION"."096P004D".SCADA := FALSE;
   END_IF;
   #_w2 := %DB78.DBX147.1 AND NOT "Tag_21";   // rising edge of %DB78.DBX147.1
   "Tag_21" := %DB78.DBX147.1;
   IF #_w2 THEN
       "MODO OPERACION"."096P004D".AUTOMATICO := TRUE;
       "MODO OPERACION"."096P004D".MANUAL := FALSE;
       "MODO OPERACION"."096P004D".SCADA := FALSE;
   END_IF;
   #_w3 := %DB78.DBX147.2 AND NOT "Tag_22";   // rising edge of %DB78.DBX147.2
   "Tag_22" := %DB78.DBX147.2;
   IF #_w3 THEN
       "MODO OPERACION"."096P004D".SCADA := TRUE;
       "MODO OPERACION"."096P004D".AUTOMATICO := FALSE;
       "MODO OPERACION"."096P004D".MANUAL := FALSE;
   END_IF;
END_REGION

REGION Network 12: estados modos de operacion
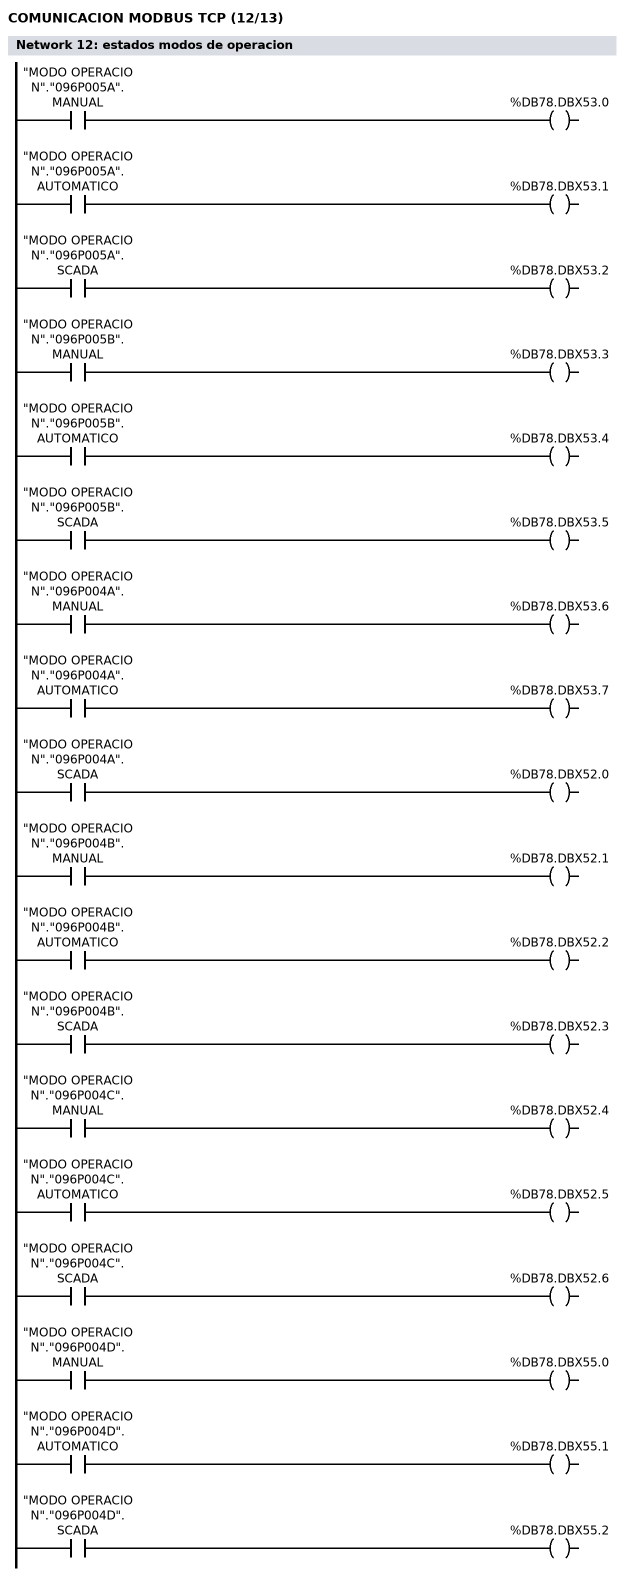
   RUNG wire#powerrail
      Contact( "MODO OPERACION"."096P005A".MANUAL )
      Coil( %DB78.DBX53.0 )
   END_RUNG
   RUNG wire#powerrail
      Contact( "MODO OPERACION"."096P005A".AUTOMATICO )
      Coil( %DB78.DBX53.1 )
   END_RUNG
   RUNG wire#powerrail
      Contact( "MODO OPERACION"."096P005A".SCADA )
      Coil( %DB78.DBX53.2 )
   END_RUNG
   RUNG wire#powerrail
      Contact( "MODO OPERACION"."096P005B".MANUAL )
      Coil( %DB78.DBX53.3 )
   END_RUNG
   RUNG wire#powerrail
      Contact( "MODO OPERACION"."096P005B".AUTOMATICO )
      Coil( %DB78.DBX53.4 )
   END_RUNG
   RUNG wire#powerrail
      Contact( "MODO OPERACION"."096P005B".SCADA )
      Coil( %DB78.DBX53.5 )
   END_RUNG
   RUNG wire#powerrail
      Contact( "MODO OPERACION"."096P004A".MANUAL )
      Coil( %DB78.DBX53.6 )
   END_RUNG
   RUNG wire#powerrail
      Contact( "MODO OPERACION"."096P004A".AUTOMATICO )
      Coil( %DB78.DBX53.7 )
   END_RUNG
   RUNG wire#powerrail
      Contact( "MODO OPERACION"."096P004A".SCADA )
      Coil( %DB78.DBX52.0 )
   END_RUNG
   RUNG wire#powerrail
      Contact( "MODO OPERACION"."096P004B".MANUAL )
      Coil( %DB78.DBX52.1 )
   END_RUNG
   RUNG wire#powerrail
      Contact( "MODO OPERACION"."096P004B".AUTOMATICO )
      Coil( %DB78.DBX52.2 )
   END_RUNG
   RUNG wire#powerrail
      Contact( "MODO OPERACION"."096P004B".SCADA )
      Coil( %DB78.DBX52.3 )
   END_RUNG
   RUNG wire#powerrail
      Contact( "MODO OPERACION"."096P004C".MANUAL )
      Coil( %DB78.DBX52.4 )
   END_RUNG
   RUNG wire#powerrail
      Contact( "MODO OPERACION"."096P004C".AUTOMATICO )
      Coil( %DB78.DBX52.5 )
   END_RUNG
   RUNG wire#powerrail
      Contact( "MODO OPERACION"."096P004C".SCADA )
      Coil( %DB78.DBX52.6 )
   END_RUNG
   RUNG wire#powerrail
      Contact( "MODO OPERACION"."096P004D".MANUAL )
      Coil( %DB78.DBX55.0 )
   END_RUNG
   RUNG wire#powerrail
      Contact( "MODO OPERACION"."096P004D".AUTOMATICO )
      Coil( %DB78.DBX55.1 )
   END_RUNG
   RUNG wire#powerrail
      Contact( "MODO OPERACION"."096P004D".SCADA )
      Coil( %DB78.DBX55.2 )
   END_RUNG
   // the same network as SCL:
   %DB78.DBX53.0 := "MODO OPERACION"."096P005A".MANUAL;
   %DB78.DBX53.1 := "MODO OPERACION"."096P005A".AUTOMATICO;
   %DB78.DBX53.2 := "MODO OPERACION"."096P005A".SCADA;
   %DB78.DBX53.3 := "MODO OPERACION"."096P005B".MANUAL;
   %DB78.DBX53.4 := "MODO OPERACION"."096P005B".AUTOMATICO;
   %DB78.DBX53.5 := "MODO OPERACION"."096P005B".SCADA;
   %DB78.DBX53.6 := "MODO OPERACION"."096P004A".MANUAL;
   %DB78.DBX53.7 := "MODO OPERACION"."096P004A".AUTOMATICO;
   %DB78.DBX52.0 := "MODO OPERACION"."096P004A".SCADA;
   %DB78.DBX52.1 := "MODO OPERACION"."096P004B".MANUAL;
   %DB78.DBX52.2 := "MODO OPERACION"."096P004B".AUTOMATICO;
   %DB78.DBX52.3 := "MODO OPERACION"."096P004B".SCADA;
   %DB78.DBX52.4 := "MODO OPERACION"."096P004C".MANUAL;
   %DB78.DBX52.5 := "MODO OPERACION"."096P004C".AUTOMATICO;
   %DB78.DBX52.6 := "MODO OPERACION"."096P004C".SCADA;
   %DB78.DBX55.0 := "MODO OPERACION"."096P004D".MANUAL;
   %DB78.DBX55.1 := "MODO OPERACION"."096P004D".AUTOMATICO;
   %DB78.DBX55.2 := "MODO OPERACION"."096P004D".SCADA;
END_REGION

REGION Network 13: ESTADO VFDS
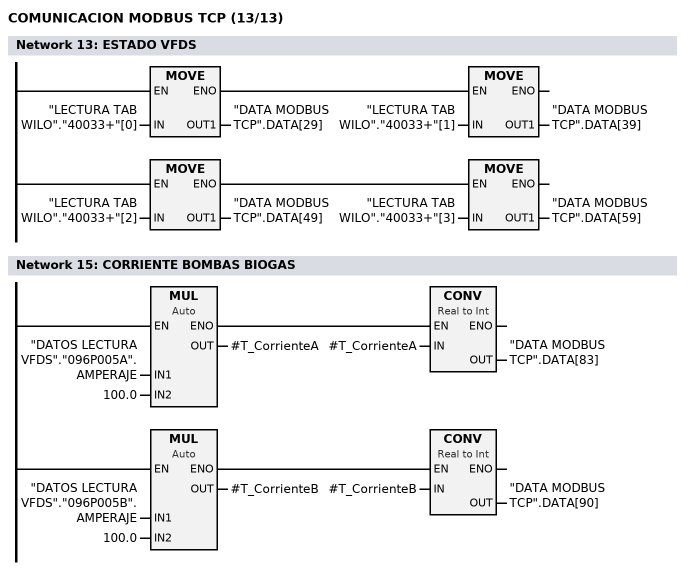
   RUNG wire#powerrail
      Move(in := "LECTURA TAB WILO"."40033+"[0], out1 => "DATA MODBUS TCP".DATA[29])
      Move(in := "LECTURA TAB WILO"."40033+"[1], out1 => "DATA MODBUS TCP".DATA[39])
   END_RUNG
   RUNG wire#powerrail
      Move(in := "LECTURA TAB WILO"."40033+"[2], out1 => "DATA MODBUS TCP".DATA[49])
      Move(in := "LECTURA TAB WILO"."40033+"[3], out1 => "DATA MODBUS TCP".DATA[59])
   END_RUNG
   // the same network as SCL:
   "DATA MODBUS TCP".DATA[29] := "LECTURA TAB WILO"."40033+"[0];
   "DATA MODBUS TCP".DATA[39] := "LECTURA TAB WILO"."40033+"[1];
   "DATA MODBUS TCP".DATA[49] := "LECTURA TAB WILO"."40033+"[2];
   "DATA MODBUS TCP".DATA[59] := "LECTURA TAB WILO"."40033+"[3];
END_REGION

REGION Network 15: CORRIENTE BOMBAS BIOGAS
   RUNG wire#powerrail
      Mul(in1 := "DATOS LECTURA VFDS"."096P005A".AMPERAJE, in2 := 100.0, out => #T_CorrienteA)
      { S7_Templates := "[SrcType := Real, DestType := Int]" } Convert(in := #T_CorrienteA, out => "DATA MODBUS TCP".DATA[83])
   END_RUNG
   RUNG wire#powerrail
      Mul(in1 := "DATOS LECTURA VFDS"."096P005B".AMPERAJE, in2 := 100.0, out => #T_CorrienteB)
      { S7_Templates := "[SrcType := Real, DestType := Int]" } Convert(in := #T_CorrienteB, out => "DATA MODBUS TCP".DATA[90])
   END_RUNG
   // the same network as SCL:
   #T_CorrienteA := "DATOS LECTURA VFDS"."096P005A".AMPERAJE * 100.0;
   "DATA MODBUS TCP".DATA[83] := REAL_TO_INT(#T_CorrienteA);
   #T_CorrienteB := "DATOS LECTURA VFDS"."096P005B".AMPERAJE * 100.0;
   "DATA MODBUS TCP".DATA[90] := REAL_TO_INT(#T_CorrienteB);
END_REGION
END_FUNCTION

FUNCTION "Comunicacion RTU" : Void   // FC8, LAD
{ S7_Optimized_Access := 'TRUE' }
VERSION : 0.1
   VAR_TEMP
      "RESET TEMP" : Bool;
      TEST1 : Bool;
   END_VAR
BEGIN

REGION Network 1: CONTEO COMUNICACION
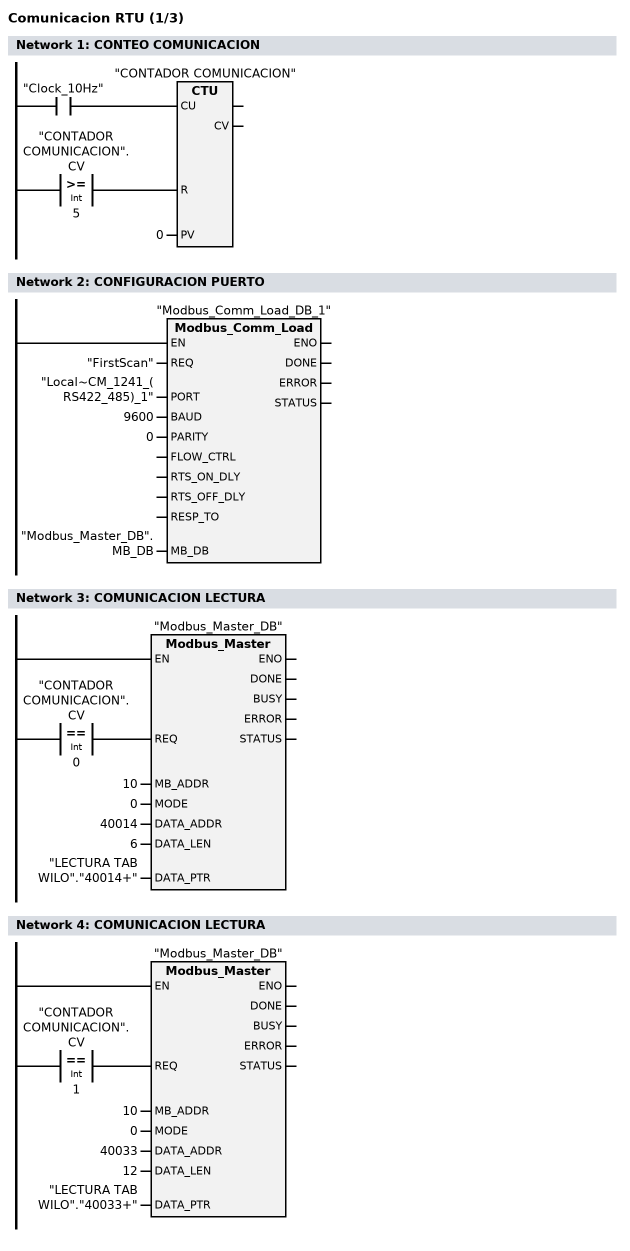
   "CONTADOR COMUNICACION".CTU(CU := "Clock_10Hz", R := "CONTADOR COMUNICACION".CV >= 5, PV := 0);
END_REGION

REGION Network 2: CONFIGURACION PUERTO
   "Modbus_Comm_Load_DB_1"(REQ := "FirstScan",   // Modbus_Comm_Load
                           PORT := "Local~CM_1241_(RS422_485)_1",
                           BAUD := 9600,
                           PARITY := 0,
                           MB_DB := "Modbus_Master_DB".MB_DB);
END_REGION

REGION Network 3: COMUNICACION LECTURA
   "Modbus_Master_DB"(REQ := "CONTADOR COMUNICACION".CV = 0,   // Modbus_Master
                      MB_ADDR := 10,
                      MODE := 0,
                      DATA_ADDR := 40014,
                      DATA_LEN := 6,
                      DATA_PTR := "LECTURA TAB WILO"."40014+");
END_REGION

REGION Network 4: COMUNICACION LECTURA
   "Modbus_Master_DB"(REQ := "CONTADOR COMUNICACION".CV = 1,   // Modbus_Master
                      MB_ADDR := 10,
                      MODE := 0,
                      DATA_ADDR := 40033,
                      DATA_LEN := 12,
                      DATA_PTR := "LECTURA TAB WILO"."40033+");
END_REGION

REGION Network 5: COMUNICACION LECTURA
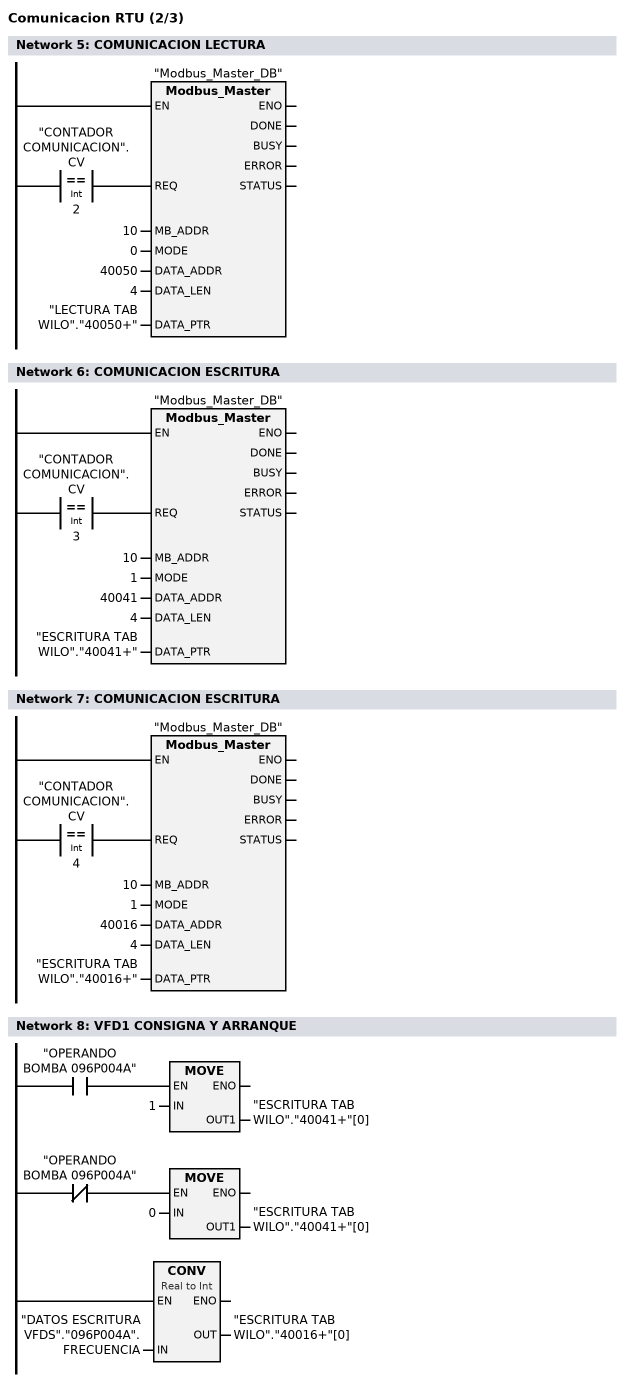
   "Modbus_Master_DB"(REQ := "CONTADOR COMUNICACION".CV = 2,   // Modbus_Master
                      MB_ADDR := 10,
                      MODE := 0,
                      DATA_ADDR := 40050,
                      DATA_LEN := 4,
                      DATA_PTR := "LECTURA TAB WILO"."40050+");
END_REGION

REGION Network 6: COMUNICACION ESCRITURA
   "Modbus_Master_DB"(REQ := "CONTADOR COMUNICACION".CV = 3,   // Modbus_Master
                      MB_ADDR := 10,
                      MODE := 1,
                      DATA_ADDR := 40041,
                      DATA_LEN := 4,
                      DATA_PTR := "ESCRITURA TAB WILO"."40041+");
END_REGION

REGION Network 7: COMUNICACION ESCRITURA
   "Modbus_Master_DB"(REQ := "CONTADOR COMUNICACION".CV = 4,   // Modbus_Master
                      MB_ADDR := 10,
                      MODE := 1,
                      DATA_ADDR := 40016,
                      DATA_LEN := 4,
                      DATA_PTR := "ESCRITURA TAB WILO"."40016+");
END_REGION

REGION Network 8: VFD1 CONSIGNA Y ARRANQUE
   RUNG wire#powerrail
      Contact( "OPERANDO BOMBA 096P004A" )
      Move(in := 1, out1 => "ESCRITURA TAB WILO"."40041+"[0])
   END_RUNG
   RUNG wire#powerrail
      I_Contact( "OPERANDO BOMBA 096P004A" )
      Move(in := 0, out1 => "ESCRITURA TAB WILO"."40041+"[0])
   END_RUNG
   RUNG wire#powerrail
      { S7_Templates := "[SrcType := Real, DestType := Int]" } Convert(in := "DATOS ESCRITURA VFDS"."096P004A".FRECUENCIA, out => "ESCRITURA TAB WILO"."40016+"[0])
   END_RUNG
   // the same network as SCL:
   IF "OPERANDO BOMBA 096P004A" THEN "ESCRITURA TAB WILO"."40041+"[0] := 1; END_IF;
   IF NOT "OPERANDO BOMBA 096P004A" THEN "ESCRITURA TAB WILO"."40041+"[0] := 0; END_IF;
   "ESCRITURA TAB WILO"."40016+"[0] := REAL_TO_INT("DATOS ESCRITURA VFDS"."096P004A".FRECUENCIA);
END_REGION

REGION Network 9: VFD2 CONSIGNA Y ARRANQUE
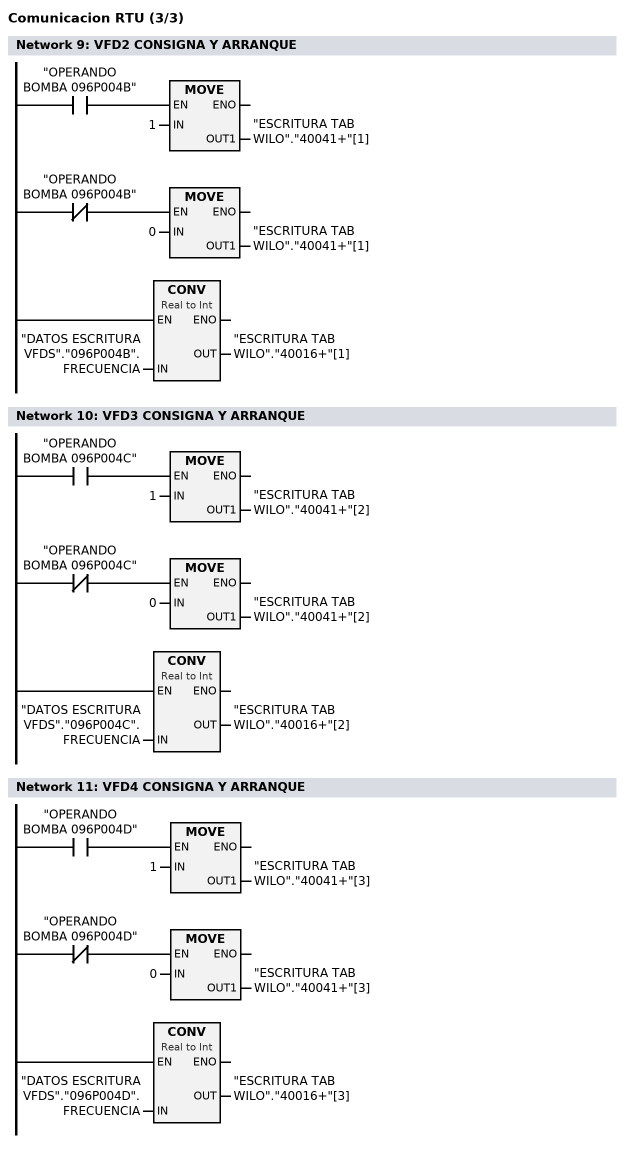
   RUNG wire#powerrail
      Contact( "OPERANDO BOMBA 096P004B" )
      Move(in := 1, out1 => "ESCRITURA TAB WILO"."40041+"[1])
   END_RUNG
   RUNG wire#powerrail
      I_Contact( "OPERANDO BOMBA 096P004B" )
      Move(in := 0, out1 => "ESCRITURA TAB WILO"."40041+"[1])
   END_RUNG
   RUNG wire#powerrail
      { S7_Templates := "[SrcType := Real, DestType := Int]" } Convert(in := "DATOS ESCRITURA VFDS"."096P004B".FRECUENCIA, out => "ESCRITURA TAB WILO"."40016+"[1])
   END_RUNG
   // the same network as SCL:
   IF "OPERANDO BOMBA 096P004B" THEN "ESCRITURA TAB WILO"."40041+"[1] := 1; END_IF;
   IF NOT "OPERANDO BOMBA 096P004B" THEN "ESCRITURA TAB WILO"."40041+"[1] := 0; END_IF;
   "ESCRITURA TAB WILO"."40016+"[1] := REAL_TO_INT("DATOS ESCRITURA VFDS"."096P004B".FRECUENCIA);
END_REGION

REGION Network 10: VFD3 CONSIGNA Y ARRANQUE
   RUNG wire#powerrail
      Contact( "OPERANDO BOMBA 096P004C" )
      Move(in := 1, out1 => "ESCRITURA TAB WILO"."40041+"[2])
   END_RUNG
   RUNG wire#powerrail
      I_Contact( "OPERANDO BOMBA 096P004C" )
      Move(in := 0, out1 => "ESCRITURA TAB WILO"."40041+"[2])
   END_RUNG
   RUNG wire#powerrail
      { S7_Templates := "[SrcType := Real, DestType := Int]" } Convert(in := "DATOS ESCRITURA VFDS"."096P004C".FRECUENCIA, out => "ESCRITURA TAB WILO"."40016+"[2])
   END_RUNG
   // the same network as SCL:
   IF "OPERANDO BOMBA 096P004C" THEN "ESCRITURA TAB WILO"."40041+"[2] := 1; END_IF;
   IF NOT "OPERANDO BOMBA 096P004C" THEN "ESCRITURA TAB WILO"."40041+"[2] := 0; END_IF;
   "ESCRITURA TAB WILO"."40016+"[2] := REAL_TO_INT("DATOS ESCRITURA VFDS"."096P004C".FRECUENCIA);
END_REGION

REGION Network 11: VFD4 CONSIGNA Y ARRANQUE
   RUNG wire#powerrail
      Contact( "OPERANDO BOMBA 096P004D" )
      Move(in := 1, out1 => "ESCRITURA TAB WILO"."40041+"[3])
   END_RUNG
   RUNG wire#powerrail
      I_Contact( "OPERANDO BOMBA 096P004D" )
      Move(in := 0, out1 => "ESCRITURA TAB WILO"."40041+"[3])
   END_RUNG
   RUNG wire#powerrail
      { S7_Templates := "[SrcType := Real, DestType := Int]" } Convert(in := "DATOS ESCRITURA VFDS"."096P004D".FRECUENCIA, out => "ESCRITURA TAB WILO"."40016+"[3])
   END_RUNG
   // the same network as SCL:
   IF "OPERANDO BOMBA 096P004D" THEN "ESCRITURA TAB WILO"."40041+"[3] := 1; END_IF;
   IF NOT "OPERANDO BOMBA 096P004D" THEN "ESCRITURA TAB WILO"."40041+"[3] := 0; END_IF;
   "ESCRITURA TAB WILO"."40016+"[3] := REAL_TO_INT("DATOS ESCRITURA VFDS"."096P004D".FRECUENCIA);
END_REGION
END_FUNCTION

FUNCTION "DATOS HMI" : Void   // FC9, LAD
{ S7_Optimized_Access := 'TRUE' }
VERSION : 0.1
   VAR_TEMP
      "FRECUENCIA 1" : Real;
      "FRECUENCIA 2" : Real;
      "FRECUENCIA 3" : Real;
      "FRECUENCIA 4" : Real;
   END_VAR
BEGIN

REGION Network 1: VFD1
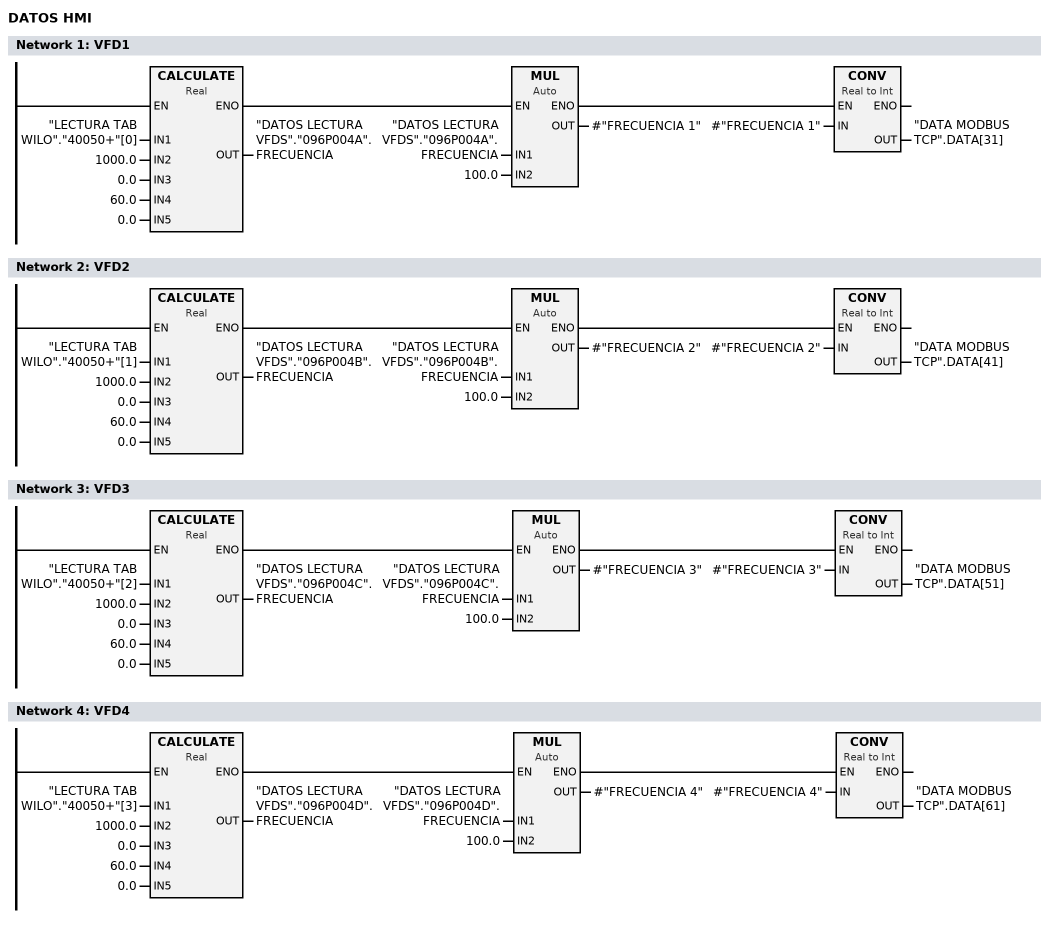
   RUNG wire#powerrail
      { S7_Templates := "SrcType := Real"; S7_Expression := "(((IN4-IN5)/(IN2-IN3))*IN1)+(IN5-(((IN4-IN5)/(IN2-IN3))*IN3))" } Calculate(in1 := "LECTURA TAB WILO"."40050+"[0], in2 := 1000.0, in3 := 0.0, in4 := 60.0, in5 := 0.0, out => "DATOS LECTURA VFDS"."096P004A".FRECUENCIA)
      Mul(in1 := "DATOS LECTURA VFDS"."096P004A".FRECUENCIA, in2 := 100.0, out => #"FRECUENCIA 1")
      { S7_Templates := "[SrcType := Real, DestType := Int]" } Convert(in := #"FRECUENCIA 1", out => "DATA MODBUS TCP".DATA[31])
   END_RUNG
   // the same network as SCL:
   "DATOS LECTURA VFDS"."096P004A".FRECUENCIA := (((60.0-0.0)/(1000.0-0.0))*"LECTURA TAB WILO"."40050+"[0])+(0.0-(((60.0-0.0)/(1000.0-0.0))*0.0));
   #"FRECUENCIA 1" := "DATOS LECTURA VFDS"."096P004A".FRECUENCIA * 100.0;
   "DATA MODBUS TCP".DATA[31] := REAL_TO_INT(#"FRECUENCIA 1");
END_REGION

REGION Network 2: VFD2
   RUNG wire#powerrail
      { S7_Templates := "SrcType := Real"; S7_Expression := "(((IN4-IN5)/(IN2-IN3))*IN1)+(IN5-(((IN4-IN5)/(IN2-IN3))*IN3))" } Calculate(in1 := "LECTURA TAB WILO"."40050+"[1], in2 := 1000.0, in3 := 0.0, in4 := 60.0, in5 := 0.0, out => "DATOS LECTURA VFDS"."096P004B".FRECUENCIA)
      Mul(in1 := "DATOS LECTURA VFDS"."096P004B".FRECUENCIA, in2 := 100.0, out => #"FRECUENCIA 2")
      { S7_Templates := "[SrcType := Real, DestType := Int]" } Convert(in := #"FRECUENCIA 2", out => "DATA MODBUS TCP".DATA[41])
   END_RUNG
   // the same network as SCL:
   "DATOS LECTURA VFDS"."096P004B".FRECUENCIA := (((60.0-0.0)/(1000.0-0.0))*"LECTURA TAB WILO"."40050+"[1])+(0.0-(((60.0-0.0)/(1000.0-0.0))*0.0));
   #"FRECUENCIA 2" := "DATOS LECTURA VFDS"."096P004B".FRECUENCIA * 100.0;
   "DATA MODBUS TCP".DATA[41] := REAL_TO_INT(#"FRECUENCIA 2");
END_REGION

REGION Network 3: VFD3
   RUNG wire#powerrail
      { S7_Templates := "SrcType := Real"; S7_Expression := "(((IN4-IN5)/(IN2-IN3))*IN1)+(IN5-(((IN4-IN5)/(IN2-IN3))*IN3))" } Calculate(in1 := "LECTURA TAB WILO"."40050+"[2], in2 := 1000.0, in3 := 0.0, in4 := 60.0, in5 := 0.0, out => "DATOS LECTURA VFDS"."096P004C".FRECUENCIA)
      Mul(in1 := "DATOS LECTURA VFDS"."096P004C".FRECUENCIA, in2 := 100.0, out => #"FRECUENCIA 3")
      { S7_Templates := "[SrcType := Real, DestType := Int]" } Convert(in := #"FRECUENCIA 3", out => "DATA MODBUS TCP".DATA[51])
   END_RUNG
   // the same network as SCL:
   "DATOS LECTURA VFDS"."096P004C".FRECUENCIA := (((60.0-0.0)/(1000.0-0.0))*"LECTURA TAB WILO"."40050+"[2])+(0.0-(((60.0-0.0)/(1000.0-0.0))*0.0));
   #"FRECUENCIA 3" := "DATOS LECTURA VFDS"."096P004C".FRECUENCIA * 100.0;
   "DATA MODBUS TCP".DATA[51] := REAL_TO_INT(#"FRECUENCIA 3");
END_REGION

REGION Network 4: VFD4
   RUNG wire#powerrail
      { S7_Templates := "SrcType := Real"; S7_Expression := "(((IN4-IN5)/(IN2-IN3))*IN1)+(IN5-(((IN4-IN5)/(IN2-IN3))*IN3))" } Calculate(in1 := "LECTURA TAB WILO"."40050+"[3], in2 := 1000.0, in3 := 0.0, in4 := 60.0, in5 := 0.0, out => "DATOS LECTURA VFDS"."096P004D".FRECUENCIA)
      Mul(in1 := "DATOS LECTURA VFDS"."096P004D".FRECUENCIA, in2 := 100.0, out => #"FRECUENCIA 4")
      { S7_Templates := "[SrcType := Real, DestType := Int]" } Convert(in := #"FRECUENCIA 4", out => "DATA MODBUS TCP".DATA[61])
   END_RUNG
   // the same network as SCL:
   "DATOS LECTURA VFDS"."096P004D".FRECUENCIA := (((60.0-0.0)/(1000.0-0.0))*"LECTURA TAB WILO"."40050+"[3])+(0.0-(((60.0-0.0)/(1000.0-0.0))*0.0));
   #"FRECUENCIA 4" := "DATOS LECTURA VFDS"."096P004D".FRECUENCIA * 100.0;
   "DATA MODBUS TCP".DATA[61] := REAL_TO_INT(#"FRECUENCIA 4");
END_REGION
END_FUNCTION

FUNCTION "FALLAS SISTEMA" : Void   // FC11, LAD
{ S7_Optimized_Access := 'TRUE' }
VERSION : 0.1
   VAR_TEMP
      "RESET 4A" : Bool;
      "RESET 4B" : Bool;
      "RESET 4C" : Bool;
      "RESET 4D" : Bool;
      "RESET 5A" : Bool;
      "RESET 5B" : Bool;
   END_VAR
BEGIN

REGION Network 1: reset gral
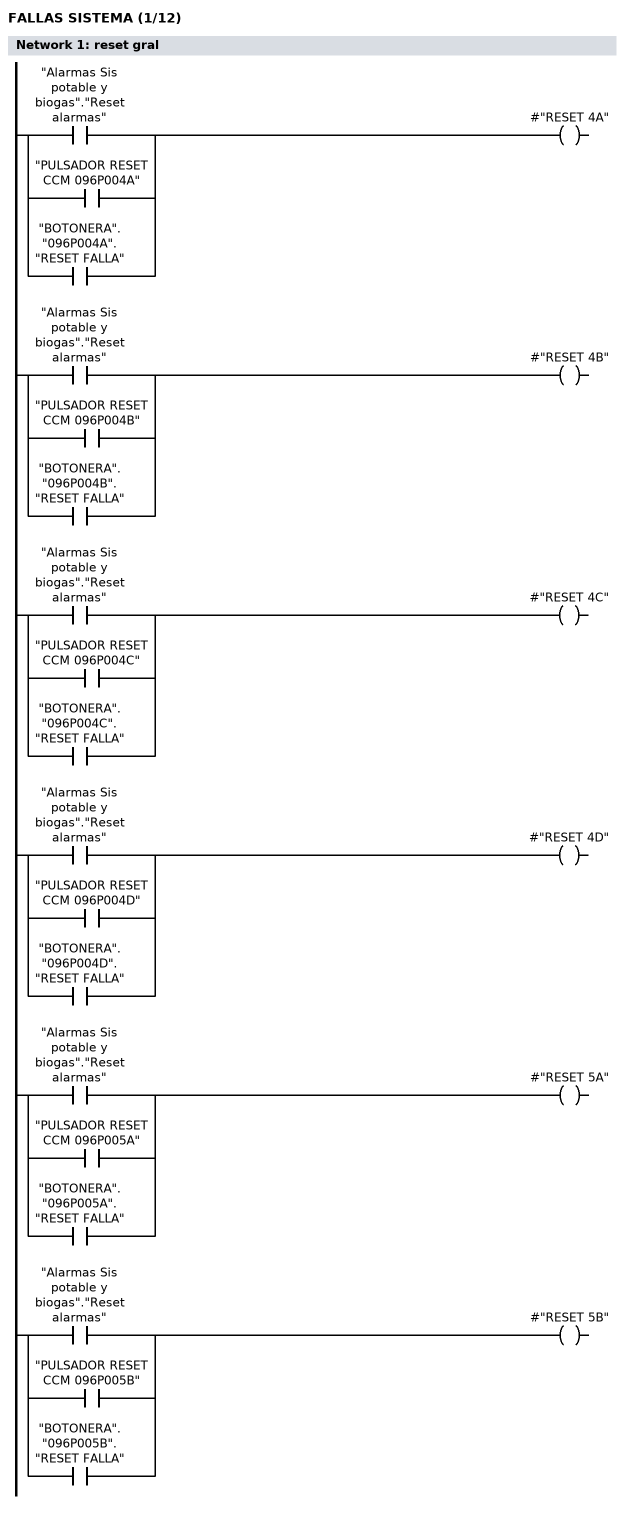
   RUNG wire#powerrail
      Contact( "Alarmas Sis potable y biogas"."Reset alarmas" )
      wire#w1
      Coil( #"RESET 4A" )
   END_RUNG
   RUNG wire#powerrail
      Contact( "PULSADOR RESET CCM 096P004A" )
   END_RUNG wire#w1
   RUNG wire#powerrail
      Contact( "BOTONERA"."096P004A"."RESET FALLA" )
   END_RUNG wire#w1
   RUNG wire#powerrail
      Contact( "Alarmas Sis potable y biogas"."Reset alarmas" )
      wire#w2
      Coil( #"RESET 4B" )
   END_RUNG
   RUNG wire#powerrail
      Contact( "PULSADOR RESET CCM 096P004B" )
   END_RUNG wire#w2
   RUNG wire#powerrail
      Contact( "BOTONERA"."096P004B"."RESET FALLA" )
   END_RUNG wire#w2
   RUNG wire#powerrail
      Contact( "Alarmas Sis potable y biogas"."Reset alarmas" )
      wire#w3
      Coil( #"RESET 4C" )
   END_RUNG
   RUNG wire#powerrail
      Contact( "PULSADOR RESET CCM 096P004C" )
   END_RUNG wire#w3
   RUNG wire#powerrail
      Contact( "BOTONERA"."096P004C"."RESET FALLA" )
   END_RUNG wire#w3
   RUNG wire#powerrail
      Contact( "Alarmas Sis potable y biogas"."Reset alarmas" )
      wire#w4
      Coil( #"RESET 4D" )
   END_RUNG
   RUNG wire#powerrail
      Contact( "PULSADOR RESET CCM 096P004D" )
   END_RUNG wire#w4
   RUNG wire#powerrail
      Contact( "BOTONERA"."096P004D"."RESET FALLA" )
   END_RUNG wire#w4
   RUNG wire#powerrail
      Contact( "Alarmas Sis potable y biogas"."Reset alarmas" )
      wire#w5
      Coil( #"RESET 5A" )
   END_RUNG
   RUNG wire#powerrail
      Contact( "PULSADOR RESET CCM 096P005A" )
   END_RUNG wire#w5
   RUNG wire#powerrail
      Contact( "BOTONERA"."096P005A"."RESET FALLA" )
   END_RUNG wire#w5
   RUNG wire#powerrail
      Contact( "Alarmas Sis potable y biogas"."Reset alarmas" )
      wire#w6
      Coil( #"RESET 5B" )
   END_RUNG
   RUNG wire#powerrail
      Contact( "PULSADOR RESET CCM 096P005B" )
   END_RUNG wire#w6
   RUNG wire#powerrail
      Contact( "BOTONERA"."096P005B"."RESET FALLA" )
   END_RUNG wire#w6
   // the same network as SCL:
   #"RESET 4A" := "Alarmas Sis potable y biogas"."Reset alarmas" OR "PULSADOR RESET CCM 096P004A" OR "BOTONERA"."096P004A"."RESET FALLA";
   #"RESET 4B" := "Alarmas Sis potable y biogas"."Reset alarmas" OR "PULSADOR RESET CCM 096P004B" OR "BOTONERA"."096P004B"."RESET FALLA";
   #"RESET 4C" := "Alarmas Sis potable y biogas"."Reset alarmas" OR "PULSADOR RESET CCM 096P004C" OR "BOTONERA"."096P004C"."RESET FALLA";
   #"RESET 4D" := "Alarmas Sis potable y biogas"."Reset alarmas" OR "PULSADOR RESET CCM 096P004D" OR "BOTONERA"."096P004D"."RESET FALLA";
   #"RESET 5A" := "Alarmas Sis potable y biogas"."Reset alarmas" OR "PULSADOR RESET CCM 096P005A" OR "BOTONERA"."096P005A"."RESET FALLA";
   #"RESET 5B" := "Alarmas Sis potable y biogas"."Reset alarmas" OR "PULSADOR RESET CCM 096P005B" OR "BOTONERA"."096P005B"."RESET FALLA";
END_REGION

REGION Network 2: PARO DE EMERGENCIA GRAL
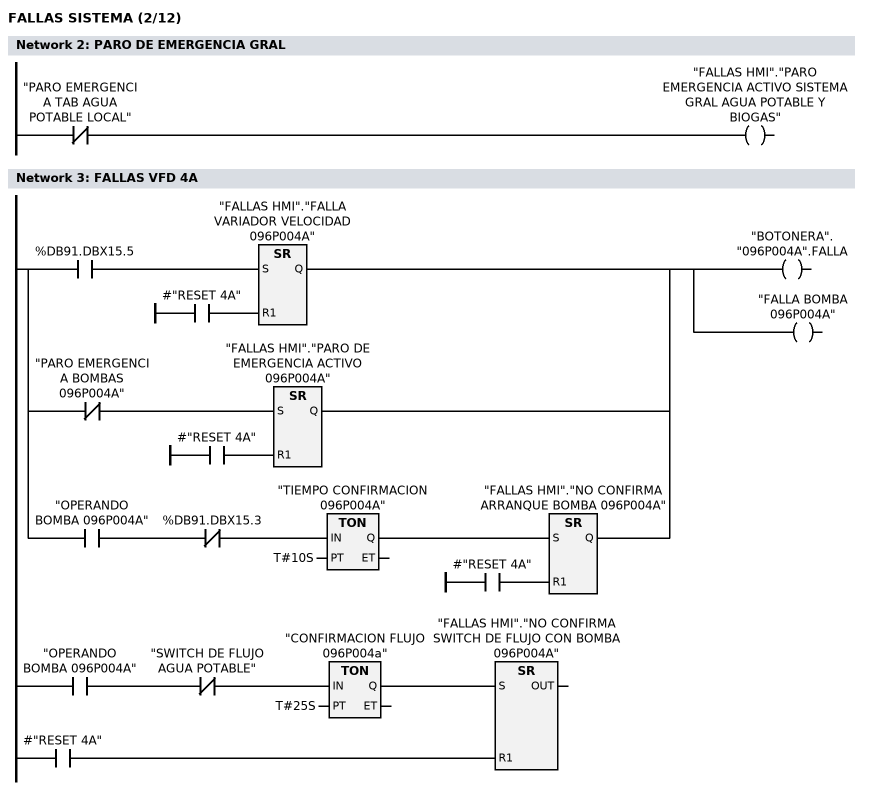
   RUNG wire#powerrail
      I_Contact( "PARO EMERGENCIA TAB AGUA POTABLE LOCAL" )
      Coil( "FALLAS HMI"."PARO EMERGENCIA ACTIVO SISTEMA GRAL AGUA POTABLE Y BIOGAS" )
   END_RUNG
   // the same network as SCL:
   "FALLAS HMI"."PARO EMERGENCIA ACTIVO SISTEMA GRAL AGUA POTABLE Y BIOGAS" := NOT "PARO EMERGENCIA TAB AGUA POTABLE LOCAL";
END_REGION

REGION Network 3: FALLAS VFD 4A
   IF %DB91.DBX15.5 THEN
       "FALLAS HMI"."FALLA VARIADOR VELOCIDAD 096P004A" := TRUE;   // SR flip-flop
   END_IF;
   IF #"RESET 4A" THEN "FALLAS HMI"."FALLA VARIADOR VELOCIDAD 096P004A" := FALSE; END_IF;
   IF NOT "PARO EMERGENCIA BOMBAS 096P004A" THEN
       "FALLAS HMI"."PARO DE EMERGENCIA ACTIVO 096P004A" := TRUE;   // SR flip-flop
   END_IF;
   IF #"RESET 4A" THEN "FALLAS HMI"."PARO DE EMERGENCIA ACTIVO 096P004A" := FALSE; END_IF;
   "TIEMPO CONFIRMACION 096P004A".TON(IN := "OPERANDO BOMBA 096P004A" AND NOT %DB91.DBX15.3, PT := T#10S);
   IF "TIEMPO CONFIRMACION 096P004A".Q THEN
       "FALLAS HMI"."NO CONFIRMA ARRANQUE BOMBA 096P004A" := TRUE;   // SR flip-flop
   END_IF;
   IF #"RESET 4A" THEN "FALLAS HMI"."NO CONFIRMA ARRANQUE BOMBA 096P004A" := FALSE; END_IF;
   "BOTONERA"."096P004A".FALLA := "FALLAS HMI"."FALLA VARIADOR VELOCIDAD 096P004A" OR "FALLAS HMI"."PARO DE EMERGENCIA ACTIVO 096P004A" OR "FALLAS HMI"."NO CONFIRMA ARRANQUE BOMBA 096P004A";
   "FALLA BOMBA 096P004A" := "BOTONERA"."096P004A".FALLA;
   "CONFIRMACION FLUJO 096P004a".TON(IN := "OPERANDO BOMBA 096P004A" AND NOT "SWITCH DE FLUJO AGUA POTABLE",
                           PT := T#25S);
   IF "CONFIRMACION FLUJO 096P004a".Q THEN
       "FALLAS HMI"."NO CONFIRMA SWITCH DE FLUJO CON BOMBA 096P004A" := TRUE;   // SR flip-flop
   END_IF;
   IF #"RESET 4A" THEN "FALLAS HMI"."NO CONFIRMA SWITCH DE FLUJO CON BOMBA 096P004A" := FALSE; END_IF;
END_REGION

REGION Network 4: FALLAS VFD 4B
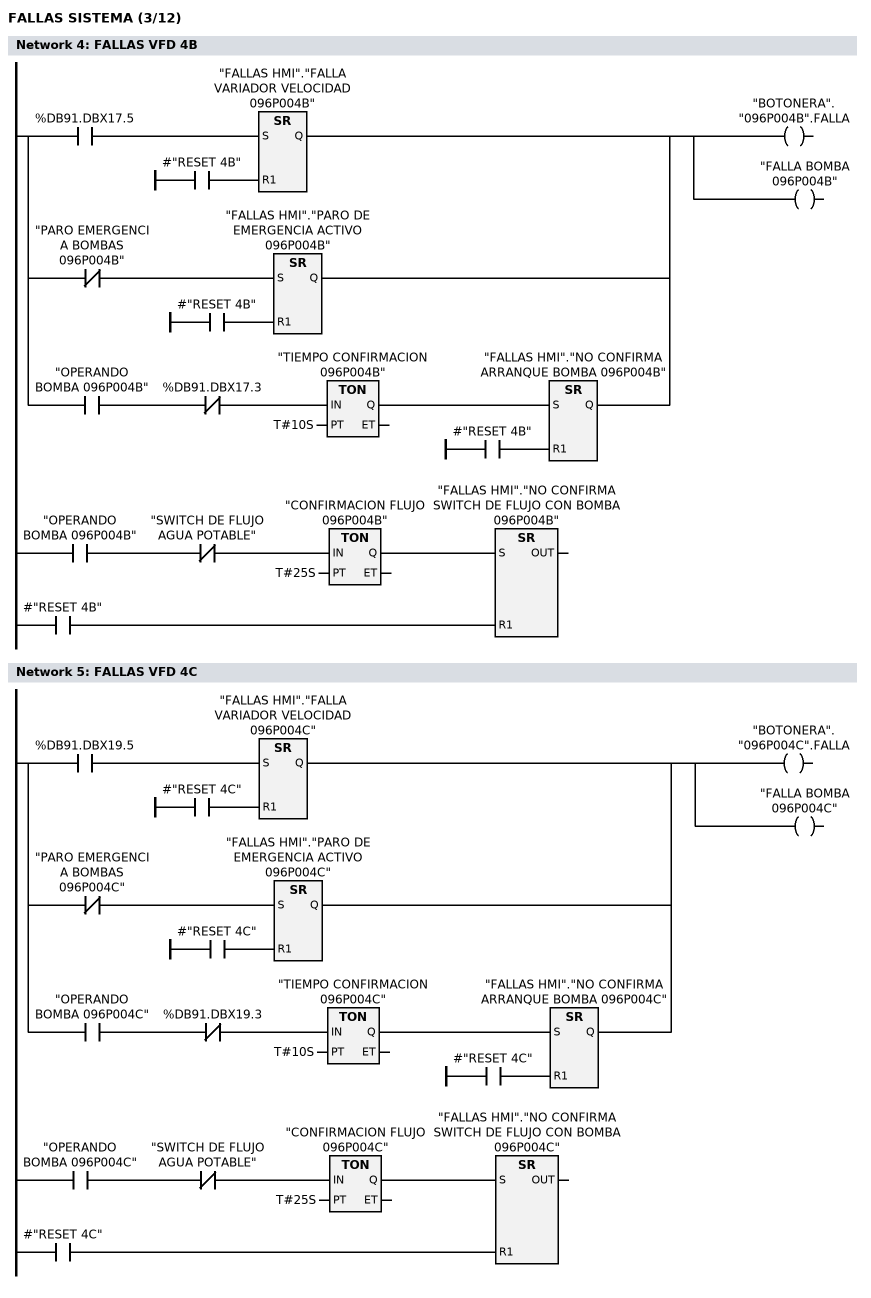
   IF %DB91.DBX17.5 THEN
       "FALLAS HMI"."FALLA VARIADOR VELOCIDAD 096P004B" := TRUE;   // SR flip-flop
   END_IF;
   IF #"RESET 4B" THEN "FALLAS HMI"."FALLA VARIADOR VELOCIDAD 096P004B" := FALSE; END_IF;
   IF NOT "PARO EMERGENCIA BOMBAS 096P004B" THEN
       "FALLAS HMI"."PARO DE EMERGENCIA ACTIVO 096P004B" := TRUE;   // SR flip-flop
   END_IF;
   IF #"RESET 4B" THEN "FALLAS HMI"."PARO DE EMERGENCIA ACTIVO 096P004B" := FALSE; END_IF;
   "TIEMPO CONFIRMACION 096P004B".TON(IN := "OPERANDO BOMBA 096P004B" AND NOT %DB91.DBX17.3, PT := T#10S);
   IF "TIEMPO CONFIRMACION 096P004B".Q THEN
       "FALLAS HMI"."NO CONFIRMA ARRANQUE BOMBA 096P004B" := TRUE;   // SR flip-flop
   END_IF;
   IF #"RESET 4B" THEN "FALLAS HMI"."NO CONFIRMA ARRANQUE BOMBA 096P004B" := FALSE; END_IF;
   "BOTONERA"."096P004B".FALLA := "FALLAS HMI"."FALLA VARIADOR VELOCIDAD 096P004B" OR "FALLAS HMI"."PARO DE EMERGENCIA ACTIVO 096P004B" OR "FALLAS HMI"."NO CONFIRMA ARRANQUE BOMBA 096P004B";
   "FALLA BOMBA 096P004B" := "BOTONERA"."096P004B".FALLA;
   "CONFIRMACION FLUJO 096P004B".TON(IN := "OPERANDO BOMBA 096P004B" AND NOT "SWITCH DE FLUJO AGUA POTABLE",
                           PT := T#25S);
   IF "CONFIRMACION FLUJO 096P004B".Q THEN
       "FALLAS HMI"."NO CONFIRMA SWITCH DE FLUJO CON BOMBA 096P004B" := TRUE;   // SR flip-flop
   END_IF;
   IF #"RESET 4B" THEN "FALLAS HMI"."NO CONFIRMA SWITCH DE FLUJO CON BOMBA 096P004B" := FALSE; END_IF;
END_REGION

REGION Network 5: FALLAS VFD 4C
   IF %DB91.DBX19.5 THEN
       "FALLAS HMI"."FALLA VARIADOR VELOCIDAD 096P004C" := TRUE;   // SR flip-flop
   END_IF;
   IF #"RESET 4C" THEN "FALLAS HMI"."FALLA VARIADOR VELOCIDAD 096P004C" := FALSE; END_IF;
   IF NOT "PARO EMERGENCIA BOMBAS 096P004C" THEN
       "FALLAS HMI"."PARO DE EMERGENCIA ACTIVO 096P004C" := TRUE;   // SR flip-flop
   END_IF;
   IF #"RESET 4C" THEN "FALLAS HMI"."PARO DE EMERGENCIA ACTIVO 096P004C" := FALSE; END_IF;
   "TIEMPO CONFIRMACION 096P004C".TON(IN := "OPERANDO BOMBA 096P004C" AND NOT %DB91.DBX19.3, PT := T#10S);
   IF "TIEMPO CONFIRMACION 096P004C".Q THEN
       "FALLAS HMI"."NO CONFIRMA ARRANQUE BOMBA 096P004C" := TRUE;   // SR flip-flop
   END_IF;
   IF #"RESET 4C" THEN "FALLAS HMI"."NO CONFIRMA ARRANQUE BOMBA 096P004C" := FALSE; END_IF;
   "BOTONERA"."096P004C".FALLA := "FALLAS HMI"."FALLA VARIADOR VELOCIDAD 096P004C" OR "FALLAS HMI"."PARO DE EMERGENCIA ACTIVO 096P004C" OR "FALLAS HMI"."NO CONFIRMA ARRANQUE BOMBA 096P004C";
   "FALLA BOMBA 096P004C" := "BOTONERA"."096P004C".FALLA;
   "CONFIRMACION FLUJO 096P004C".TON(IN := "OPERANDO BOMBA 096P004C" AND NOT "SWITCH DE FLUJO AGUA POTABLE",
                           PT := T#25S);
   IF "CONFIRMACION FLUJO 096P004C".Q THEN
       "FALLAS HMI"."NO CONFIRMA SWITCH DE FLUJO CON BOMBA 096P004C" := TRUE;   // SR flip-flop
   END_IF;
   IF #"RESET 4C" THEN "FALLAS HMI"."NO CONFIRMA SWITCH DE FLUJO CON BOMBA 096P004C" := FALSE; END_IF;
END_REGION

REGION Network 6: FALLAS VFD 4D
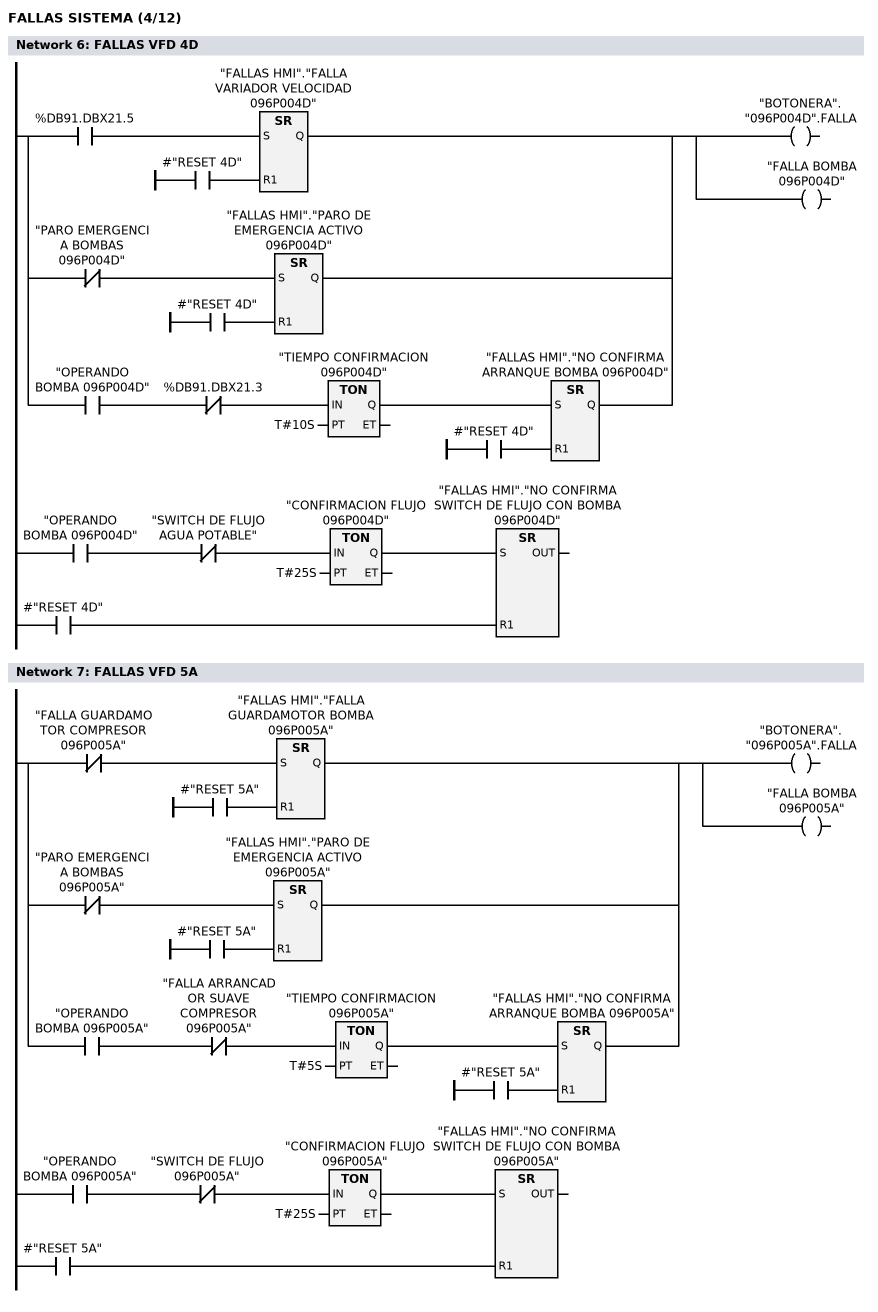
   IF %DB91.DBX21.5 THEN
       "FALLAS HMI"."FALLA VARIADOR VELOCIDAD 096P004D" := TRUE;   // SR flip-flop
   END_IF;
   IF #"RESET 4D" THEN "FALLAS HMI"."FALLA VARIADOR VELOCIDAD 096P004D" := FALSE; END_IF;
   IF NOT "PARO EMERGENCIA BOMBAS 096P004D" THEN
       "FALLAS HMI"."PARO DE EMERGENCIA ACTIVO 096P004D" := TRUE;   // SR flip-flop
   END_IF;
   IF #"RESET 4D" THEN "FALLAS HMI"."PARO DE EMERGENCIA ACTIVO 096P004D" := FALSE; END_IF;
   "TIEMPO CONFIRMACION 096P004D".TON(IN := "OPERANDO BOMBA 096P004D" AND NOT %DB91.DBX21.3, PT := T#10S);
   IF "TIEMPO CONFIRMACION 096P004D".Q THEN
       "FALLAS HMI"."NO CONFIRMA ARRANQUE BOMBA 096P004D" := TRUE;   // SR flip-flop
   END_IF;
   IF #"RESET 4D" THEN "FALLAS HMI"."NO CONFIRMA ARRANQUE BOMBA 096P004D" := FALSE; END_IF;
   "BOTONERA"."096P004D".FALLA := "FALLAS HMI"."FALLA VARIADOR VELOCIDAD 096P004D" OR "FALLAS HMI"."PARO DE EMERGENCIA ACTIVO 096P004D" OR "FALLAS HMI"."NO CONFIRMA ARRANQUE BOMBA 096P004D";
   "FALLA BOMBA 096P004D" := "BOTONERA"."096P004D".FALLA;
   "CONFIRMACION FLUJO 096P004D".TON(IN := "OPERANDO BOMBA 096P004D" AND NOT "SWITCH DE FLUJO AGUA POTABLE",
                           PT := T#25S);
   IF "CONFIRMACION FLUJO 096P004D".Q THEN
       "FALLAS HMI"."NO CONFIRMA SWITCH DE FLUJO CON BOMBA 096P004D" := TRUE;   // SR flip-flop
   END_IF;
   IF #"RESET 4D" THEN "FALLAS HMI"."NO CONFIRMA SWITCH DE FLUJO CON BOMBA 096P004D" := FALSE; END_IF;
END_REGION

REGION Network 7: FALLAS VFD 5A
   IF NOT "FALLA GUARDAMOTOR COMPRESOR 096P005A" THEN
       "FALLAS HMI"."FALLA GUARDAMOTOR BOMBA 096P005A" := TRUE;   // SR flip-flop
   END_IF;
   IF #"RESET 5A" THEN "FALLAS HMI"."FALLA GUARDAMOTOR BOMBA 096P005A" := FALSE; END_IF;
   IF NOT "PARO EMERGENCIA BOMBAS 096P005A" THEN
       "FALLAS HMI"."PARO DE EMERGENCIA ACTIVO 096P005A" := TRUE;   // SR flip-flop
   END_IF;
   IF #"RESET 5A" THEN "FALLAS HMI"."PARO DE EMERGENCIA ACTIVO 096P005A" := FALSE; END_IF;
   "TIEMPO CONFIRMACION 096P005A".TON(IN := "OPERANDO BOMBA 096P005A" AND NOT "FALLA ARRANCADOR SUAVE COMPRESOR 096P005A",
                           PT := T#5S);
   IF "TIEMPO CONFIRMACION 096P005A".Q THEN
       "FALLAS HMI"."NO CONFIRMA ARRANQUE BOMBA 096P005A" := TRUE;   // SR flip-flop
   END_IF;
   IF #"RESET 5A" THEN "FALLAS HMI"."NO CONFIRMA ARRANQUE BOMBA 096P005A" := FALSE; END_IF;
   "BOTONERA"."096P005A".FALLA := "FALLAS HMI"."FALLA GUARDAMOTOR BOMBA 096P005A" OR "FALLAS HMI"."PARO DE EMERGENCIA ACTIVO 096P005A" OR "FALLAS HMI"."NO CONFIRMA ARRANQUE BOMBA 096P005A";
   "FALLA BOMBA 096P005A" := "BOTONERA"."096P005A".FALLA;
   "CONFIRMACION FLUJO 096P005A".TON(IN := "OPERANDO BOMBA 096P005A" AND NOT "SWITCH DE FLUJO 096P005A",
                           PT := T#25S);
   IF "CONFIRMACION FLUJO 096P005A".Q THEN
       "FALLAS HMI"."NO CONFIRMA SWITCH DE FLUJO CON BOMBA 096P005A" := TRUE;   // SR flip-flop
   END_IF;
   IF #"RESET 5A" THEN "FALLAS HMI"."NO CONFIRMA SWITCH DE FLUJO CON BOMBA 096P005A" := FALSE; END_IF;
END_REGION

REGION Network 8: FALLAS VFD 5B
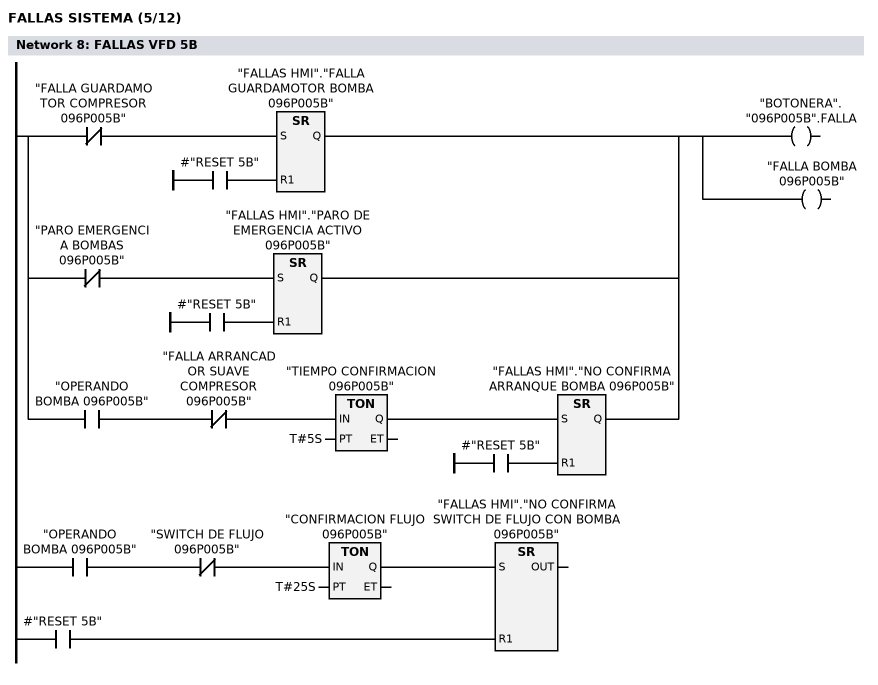
   IF NOT "FALLA GUARDAMOTOR COMPRESOR 096P005B" THEN
       "FALLAS HMI"."FALLA GUARDAMOTOR BOMBA 096P005B" := TRUE;   // SR flip-flop
   END_IF;
   IF #"RESET 5B" THEN "FALLAS HMI"."FALLA GUARDAMOTOR BOMBA 096P005B" := FALSE; END_IF;
   IF NOT "PARO EMERGENCIA BOMBAS 096P005B" THEN
       "FALLAS HMI"."PARO DE EMERGENCIA ACTIVO 096P005B" := TRUE;   // SR flip-flop
   END_IF;
   IF #"RESET 5B" THEN "FALLAS HMI"."PARO DE EMERGENCIA ACTIVO 096P005B" := FALSE; END_IF;
   "TIEMPO CONFIRMACION 096P005B".TON(IN := "OPERANDO BOMBA 096P005B" AND NOT "FALLA ARRANCADOR SUAVE COMPRESOR 096P005B",
                           PT := T#5S);
   IF "TIEMPO CONFIRMACION 096P005B".Q THEN
       "FALLAS HMI"."NO CONFIRMA ARRANQUE BOMBA 096P005B" := TRUE;   // SR flip-flop
   END_IF;
   IF #"RESET 5B" THEN "FALLAS HMI"."NO CONFIRMA ARRANQUE BOMBA 096P005B" := FALSE; END_IF;
   "BOTONERA"."096P005B".FALLA := "FALLAS HMI"."FALLA GUARDAMOTOR BOMBA 096P005B" OR "FALLAS HMI"."PARO DE EMERGENCIA ACTIVO 096P005B" OR "FALLAS HMI"."NO CONFIRMA ARRANQUE BOMBA 096P005B";
   "FALLA BOMBA 096P005B" := "BOTONERA"."096P005B".FALLA;
   "CONFIRMACION FLUJO 096P005B".TON(IN := "OPERANDO BOMBA 096P005B" AND NOT "SWITCH DE FLUJO 096P005B",
                           PT := T#25S);
   IF "CONFIRMACION FLUJO 096P005B".Q THEN
       "FALLAS HMI"."NO CONFIRMA SWITCH DE FLUJO CON BOMBA 096P005B" := TRUE;   // SR flip-flop
   END_IF;
   IF #"RESET 5B" THEN "FALLAS HMI"."NO CONFIRMA SWITCH DE FLUJO CON BOMBA 096P005B" := FALSE; END_IF;
END_REGION

REGION Network 9: FALLA BAJA PRESION EN SUCCION AGUA POTABLE
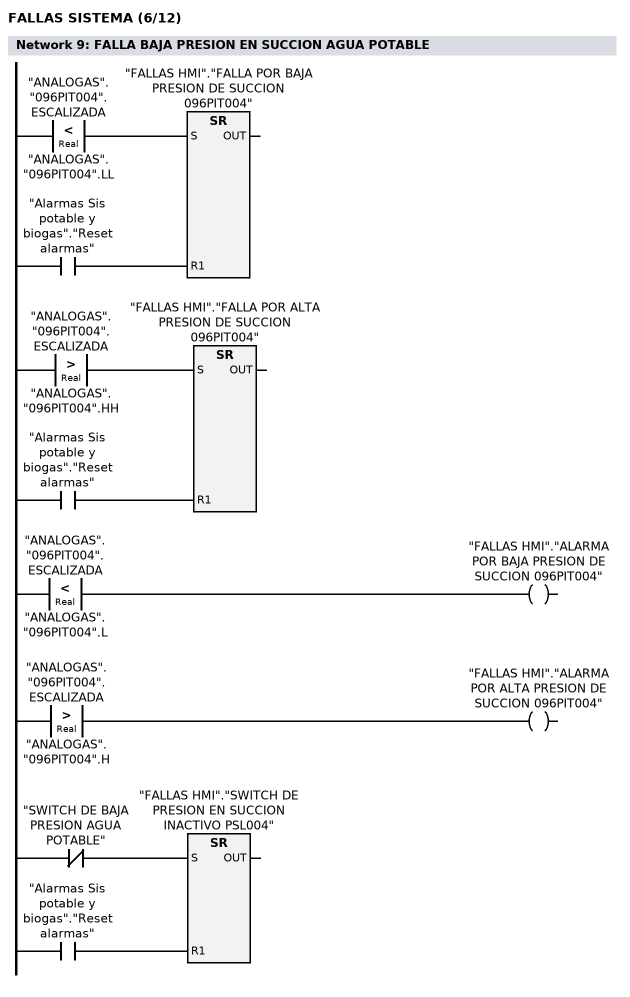
   RUNG wire#powerrail
      { S7_Templates := "SrcType := Real" } LT_Contact(in1 := "ANALOGAS"."096PIT004".ESCALIZADA, in2 := "ANALOGAS"."096PIT004".LL)
      S_SR(operand := "FALLAS HMI"."FALLA POR BAJA PRESION DE SUCCION 096PIT004", r1 := wire#w1)
   END_RUNG
   RUNG wire#powerrail
      Contact( "Alarmas Sis potable y biogas"."Reset alarmas" )
   END_RUNG wire#w1
   RUNG wire#powerrail
      { S7_Templates := "SrcType := Real" } GT_Contact(in1 := "ANALOGAS"."096PIT004".ESCALIZADA, in2 := "ANALOGAS"."096PIT004".HH)
      S_SR(operand := "FALLAS HMI"."FALLA POR ALTA PRESION DE SUCCION 096PIT004", r1 := wire#w2)
   END_RUNG
   RUNG wire#powerrail
      Contact( "Alarmas Sis potable y biogas"."Reset alarmas" )
   END_RUNG wire#w2
   RUNG wire#powerrail
      { S7_Templates := "SrcType := Real" } LT_Contact(in1 := "ANALOGAS"."096PIT004".ESCALIZADA, in2 := "ANALOGAS"."096PIT004".L)
      Coil( "FALLAS HMI"."ALARMA POR BAJA PRESION DE SUCCION 096PIT004" )
   END_RUNG
   RUNG wire#powerrail
      { S7_Templates := "SrcType := Real" } GT_Contact(in1 := "ANALOGAS"."096PIT004".ESCALIZADA, in2 := "ANALOGAS"."096PIT004".H)
      Coil( "FALLAS HMI"."ALARMA POR ALTA PRESION DE SUCCION 096PIT004" )
   END_RUNG
   RUNG wire#powerrail
      I_Contact( "SWITCH DE BAJA PRESION AGUA POTABLE" )
      S_SR(operand := "FALLAS HMI"."SWITCH DE PRESION EN SUCCION INACTIVO PSL004", r1 := wire#w3)
   END_RUNG
   RUNG wire#powerrail
      Contact( "Alarmas Sis potable y biogas"."Reset alarmas" )
   END_RUNG wire#w3
   // the same network as SCL:
   IF "ANALOGAS"."096PIT004".ESCALIZADA < "ANALOGAS"."096PIT004".LL THEN
       "FALLAS HMI"."FALLA POR BAJA PRESION DE SUCCION 096PIT004" := TRUE;   // SR flip-flop
   END_IF;
   IF "Alarmas Sis potable y biogas"."Reset alarmas" THEN
       "FALLAS HMI"."FALLA POR BAJA PRESION DE SUCCION 096PIT004" := FALSE;
   END_IF;
   IF "ANALOGAS"."096PIT004".ESCALIZADA > "ANALOGAS"."096PIT004".HH THEN
       "FALLAS HMI"."FALLA POR ALTA PRESION DE SUCCION 096PIT004" := TRUE;   // SR flip-flop
   END_IF;
   IF "Alarmas Sis potable y biogas"."Reset alarmas" THEN
       "FALLAS HMI"."FALLA POR ALTA PRESION DE SUCCION 096PIT004" := FALSE;
   END_IF;
   "FALLAS HMI"."ALARMA POR BAJA PRESION DE SUCCION 096PIT004" := "ANALOGAS"."096PIT004".ESCALIZADA < "ANALOGAS"."096PIT004".L;
   "FALLAS HMI"."ALARMA POR ALTA PRESION DE SUCCION 096PIT004" := "ANALOGAS"."096PIT004".ESCALIZADA > "ANALOGAS"."096PIT004".H;
   IF NOT "SWITCH DE BAJA PRESION AGUA POTABLE" THEN
       "FALLAS HMI"."SWITCH DE PRESION EN SUCCION INACTIVO PSL004" := TRUE;   // SR flip-flop
   END_IF;
   IF "Alarmas Sis potable y biogas"."Reset alarmas" THEN
       "FALLAS HMI"."SWITCH DE PRESION EN SUCCION INACTIVO PSL004" := FALSE;
   END_IF;
END_REGION

REGION Network 10: FALLA BAJA PRESION EN SUCCION 5A
